C07214=1045.953,107.180,-87.113,170.483,36.346,156.840
C07215=1045.947,106.931,-87.093,170.482,36.345,156.840
C07216=1045.940,106.682,-87.073,170.480,36.343,156.840
C07217=1045.935,106.432,-87.053,170.478,36.342,156.840
C07218=1045.928,106.184,-87.034,170.477,36.340,156.839
C07219=1045.922,105.935,-87.014,170.474,36.338,156.839
C07220=1045.916,105.685,-86.994,170.472,36.337,156.839
C07221=1045.910,105.436,-86.974,170.470,36.335,156.838
C07222=1045.904,105.187,-86.955,170.469,36.334,156.838
C07223=1045.898,104.938,-86.935,170.467,36.332,156.838
C07224=1045.891,104.688,-86.916,170.465,36.331,156.838
C07225=1045.885,104.439,-86.896,170.463,36.330,156.837
C07226=1045.879,104.190,-86.876,170.461,36.328,156.837
C07227=1045.873,103.941,-86.856,170.459,36.327,156.837
C07228=1045.867,103.692,-86.837,170.458,36.325,156.836
C07229=1045.860,103.443,-86.817,170.456,36.323,156.836
C07230=1045.854,103.193,-86.798,170.454,36.322,156.836
C07231=1045.848,102.944,-86.778,170.452,36.320,156.835
C07232=1045.842,102.696,-86.758,170.450,36.318,156.835
C07233=1045.837,102.446,-86.739,170.448,36.317,156.835
C07234=1045.831,102.197,-86.719,170.447,36.316,156.835
C07235=1045.823,101.948,-86.700,170.445,36.314,156.834
C07236=1045.817,101.699,-86.680,170.443,36.313,156.834
C07237=1045.812,101.449,-86.661,170.441,36.311,156.834
C07238=1045.806,101.201,-86.641,170.439,36.310,156.833
C07239=1045.800,100.951,-86.622,170.437,36.308,156.833
C07240=1045.793,100.703,-86.602,170.436,36.307,156.833
C07241=1045.787,100.452,-86.583,170.434,36.305,156.833
C07242=1045.781,100.204,-86.563,170.432,36.303,156.832
C07243=1045.775,99.955,-86.544,170.430,36.302,156.832
C07244=1045.769,99.705,-86.525,170.428,36.300,156.832
C07245=1045.762,99.457,-86.505,170.426,36.299,156.831
C07246=1045.756,99.206,-86.486,170.425,36.298,156.831
C07247=1045.750,98.958,-86.466,170.423,36.296,156.831
C07248=1045.744,98.708,-86.447,170.421,36.295,156.831
C07249=1045.738,98.459,-86.428,170.419,36.293,156.830
C07250=1045.731,98.211,-86.409,170.417,36.292,156.830
C07251=1045.725,97.961,-86.389,170.415,36.290,156.830
C07252=1045.719,97.712,-86.371,170.413,36.289,156.830
C07253=1045.712,97.462,-86.350,170.412,36.287,156.829
C07254=1045.706,97.213,-86.332,170.410,36.286,156.829
C07255=1045.700,96.965,-86.312,170.408,36.284,156.829
C07256=1045.694,96.715,-86.293,170.406,36.283,156.828
C07257=1045.688,96.466,-86.274,170.404,36.282,156.828
C07258=1045.682,96.217,-86.255,170.402,36.280,156.828
C07259=1045.675,95.968,-86.235,170.401,36.278,156.828
C07260=1045.670,95.719,-86.216,170.399,36.277,156.827
C07261=1045.663,95.469,-86.197,170.397,36.275,156.827
C07262=1045.657,95.220,-86.177,170.395,36.274,156.827
C07263=1045.650,94.971,-86.158,170.393,36.273,156.827
C07264=1045.645,94.721,-86.139,170.391,36.271,156.826
C07265=1045.638,94.472,-86.121,170.390,36.270,156.826
C07266=1045.632,94.224,-86.101,170.388,36.268,156.826
C07267=1045.626,93.974,-86.082,170.386,36.266,156.825
C07268=1045.618,93.627,-86.055,170.383,36.265,156.825
C07269=1045.609,93.280,-86.028,170.381,36.262,156.824
C07270=1045.600,92.933,-86.001,170.378,36.260,156.824
C07271=1045.592,92.585,-85.975,170.376,36.258,156.824
C07272=1045.586,92.337,-85.955,170.374,36.256,156.823
C07273=1045.580,92.087,-85.937,170.372,36.255,156.823
C07274=1045.574,91.838,-85.918,170.370,36.254,156.823
C07275=1045.567,91.589,-85.899,170.368,36.252,156.823
C07276=1045.562,91.339,-85.880,170.367,36.251,156.822
C07277=1045.555,91.090,-85.861,170.365,36.249,156.822
C07278=1045.549,90.841,-85.841,170.363,36.248,156.822
C07279=1045.543,90.592,-85.822,170.362,36.246,156.822
C07280=1045.537,90.343,-85.803,170.359,36.245,156.821
C07281=1045.531,90.094,-85.784,170.357,36.243,156.821
C07282=1045.524,89.845,-85.766,170.356,36.242,156.821
C07283=1045.518,89.596,-85.747,170.354,36.240,156.820
C07284=1045.512,89.345,-85.728,170.352,36.239,156.820
C07285=1045.505,89.096,-85.709,170.351,36.238,156.820
C07286=1045.499,88.847,-85.690,170.349,36.236,156.820
C07287=1045.493,88.598,-85.671,170.346,36.234,156.819
C07288=1045.487,88.349,-85.652,170.345,36.233,156.819
C07289=1045.480,88.099,-85.634,170.343,36.232,156.819
C07290=1045.474,87.850,-85.615,170.341,36.231,156.819
C07291=1045.467,87.601,-85.596,170.340,36.229,156.818
C07292=1045.462,87.352,-85.577,170.338,36.228,156.818
C07293=1045.455,87.103,-85.559,170.335,36.226,156.818
C07294=1045.449,86.854,-85.540,170.334,36.224,156.817
C07295=1045.442,86.604,-85.521,170.332,36.223,156.817
C07296=1045.437,86.355,-85.502,170.330,36.222,156.817
C07297=1045.430,86.106,-85.483,170.329,36.221,156.817
C07298=1045.424,85.857,-85.465,170.327,36.219,156.816
C07299=1045.418,85.608,-85.446,170.325,36.217,156.816
C07300=1045.412,85.358,-85.427,170.323,36.216,156.816
C07301=1045.405,85.109,-85.408,170.321,36.214,156.816
C07302=1045.399,84.860,-85.390,170.319,36.213,156.815
C07303=1045.393,84.611,-85.371,170.318,36.212,156.815
C07304=1045.387,84.361,-85.352,170.316,36.211,156.815
C07305=1045.380,84.112,-85.333,170.314,36.209,156.815
C07306=1045.374,83.863,-85.315,170.313,36.207,156.814
C07307=1045.368,83.614,-85.297,170.310,36.206,156.814
C07308=1045.362,83.365,-85.278,170.308,36.204,156.814
C07309=1045.356,83.116,-85.259,170.307,36.203,156.813
C07310=1045.350,82.866,-85.240,170.305,36.202,156.813
C07311=1045.344,82.617,-85.222,170.303,36.200,156.813
C07312=1045.337,82.368,-85.203,170.302,36.199,156.813
C07313=1045.331,82.118,-85.185,170.300,36.197,156.812
C07314=1045.325,81.869,-85.166,170.297,36.195,156.812
C07315=1045.319,81.620,-85.147,170.296,36.194,156.812
C07316=1045.312,81.371,-85.128,170.294,36.193,156.812
C07317=1045.306,81.122,-85.110,170.292,36.192,156.811
C07318=1045.300,80.873,-85.091,170.291,36.190,156.811
C07319=1045.295,80.623,-85.073,170.289,36.188,156.811
C07320=1045.288,80.374,-85.054,170.288,36.187,156.811
C07321=1045.282,80.125,-85.036,170.285,36.185,156.810
C07322=1045.276,79.876,-85.017,170.283,36.184,156.810
C07323=1045.269,79.626,-84.999,170.282,36.183,156.810
C07324=1045.264,79.408,-84.982,170.280,36.181,156.809
C07325=1045.259,79.189,-84.966,170.279,36.180,156.809
C07326=1045.254,78.971,-84.950,170.277,36.178,156.809
C07327=1045.248,78.752,-84.934,170.275,36.177,156.809
C07328=1045.243,78.533,-84.917,170.273,36.176,156.808
C07329=1045.237,78.314,-84.901,170.272,36.175,156.808
C07330=1045.231,78.096,-84.885,170.270,36.173,156.808
C07331=1045.227,77.877,-84.869,170.269,36.172,156.808
C07332=1045.219,77.591,-84.848,170.267,36.171,156.807
C07333=1045.212,77.306,-84.827,170.265,36.169,156.807
C07334=1045.205,77.019,-84.806,170.263,36.168,156.807
C07335=1045.198,76.733,-84.785,170.260,36.166,156.807
C07336=1045.192,76.484,-84.766,170.259,36.164,156.806
C07337=1045.185,76.235,-84.748,170.257,36.163,156.806
C07338=1045.179,75.985,-84.730,170.255,36.161,156.806
C07339=1045.173,75.736,-84.711,170.254,36.160,156.805
C07340=1045.167,75.487,-84.693,170.252,36.159,156.805
C07341=1045.160,75.237,-84.675,170.250,36.158,156.805
C07342=1045.154,74.988,-84.657,170.248,36.156,156.805
C07343=1045.148,74.739,-84.638,170.246,36.154,156.804
C07344=1045.142,74.490,-84.620,170.244,36.153,156.804
C07345=1045.135,74.241,-84.602,170.243,36.152,156.804
C07346=1045.129,73.992,-84.584,170.241,36.151,156.804
C07347=1045.122,73.742,-84.566,170.239,36.149,156.803
C07348=1045.117,73.494,-84.548,170.238,36.147,156.803
C07349=1045.111,73.244,-84.530,170.235,36.146,156.803
C07350=1045.104,72.995,-84.511,170.233,36.145,156.803
C07351=1045.098,72.745,-84.493,170.232,36.143,156.802
C07352=1045.092,72.496,-84.474,170.230,36.142,156.802
C07353=1045.085,72.246,-84.456,170.228,36.140,156.802
C07354=1045.080,71.998,-84.438,170.227,36.139,156.802
C07355=1045.073,71.748,-84.420,170.225,36.137,156.801
C07356=1045.067,71.499,-84.402,170.222,36.136,156.801
C07357=1045.060,71.249,-84.384,170.221,36.135,156.801
C07358=1045.054,71.001,-84.366,170.219,36.134,156.801
C07359=1045.048,70.751,-84.348,170.217,36.132,156.800
C07360=1045.042,70.502,-84.329,170.216,36.130,156.800
C07361=1045.036,70.252,-84.311,170.214,36.129,156.800
C07362=1045.030,70.003,-84.294,170.213,36.128,156.800
C07363=1045.024,69.754,-84.275,170.210,36.126,156.799
C07364=1045.018,69.504,-84.257,170.208,36.125,156.799
C07365=1045.010,69.256,-84.239,170.207,36.123,156.799
C07366=1045.004,69.006,-84.221,170.205,36.122,156.799
C07367=1044.999,68.757,-84.204,170.203,36.121,156.798
C07368=1044.992,68.508,-84.185,170.202,36.119,156.798
C07369=1044.986,68.258,-84.168,170.200,36.118,156.798
C07370=1044.979,68.009,-84.150,170.197,36.116,156.797
C07371=1044.974,67.760,-84.132,170.196,36.115,156.797
C07372=1044.967,67.510,-84.114,170.194,36.114,156.797
C07373=1044.961,67.261,-84.096,170.192,36.112,156.797
C07374=1044.954,67.012,-84.078,170.191,36.111,156.796
C07375=1044.949,66.763,-84.060,170.189,36.109,156.796
C07376=1044.943,66.513,-84.042,170.187,36.108,156.796
C07377=1044.935,66.264,-84.024,170.186,36.107,156.796
C07378=1044.930,66.015,-84.006,170.183,36.106,156.795
C07379=1044.924,65.765,-83.989,170.181,36.104,156.795
C07380=1044.917,65.516,-83.971,170.180,36.102,156.795
C07381=1044.910,65.267,-83.953,170.178,36.101,156.795
C07382=1044.905,65.018,-83.935,170.176,36.100,156.794
C07383=1044.898,64.768,-83.918,170.174,36.099,156.794
C07384=1044.892,64.519,-83.900,170.173,36.097,156.794
C07385=1044.886,64.270,-83.881,170.170,36.095,156.794
C07386=1044.880,64.020,-83.864,170.168,36.094,156.793
C07387=1044.873,63.771,-83.846,170.167,36.093,156.793
C07388=1044.866,63.522,-83.829,170.165,36.092,156.793
C07389=1044.861,63.273,-83.811,170.163,36.090,156.793
C07390=1044.854,63.023,-83.794,170.162,36.089,156.792
C07391=1044.848,62.773,-83.776,170.160,36.088,156.792
C07392=1044.841,62.525,-83.758,170.158,36.087,156.792
C07393=1044.835,62.276,-83.740,170.156,36.085,156.792
C07394=1044.828,62.026,-83.723,170.154,36.084,156.792
C07395=1044.822,61.776,-83.705,170.152,36.083,156.791
C07396=1044.814,61.491,-83.686,170.150,36.081,156.791
C07397=1044.807,61.204,-83.665,170.148,36.080,156.791
C07398=1044.800,60.918,-83.645,170.146,36.078,156.791
C07399=1044.792,60.632,-83.625,170.144,36.076,156.790
C07400=1044.787,60.383,-83.608,170.142,36.075,156.790
C07401=1044.780,60.133,-83.590,170.140,36.074,156.790
C07402=1044.773,59.884,-83.573,170.138,36.073,156.789
C07403=1044.768,59.635,-83.555,170.137,36.071,156.789
C07404=1044.760,59.386,-83.537,170.135,36.070,156.789
C07405=1044.754,59.136,-83.519,170.133,36.069,156.789
C07406=1044.748,58.887,-83.502,170.132,36.067,156.789
C07407=1044.742,58.638,-83.484,170.130,36.066,156.788
C07408=1044.735,58.388,-83.467,170.128,36.065,156.788
C07409=1044.729,58.139,-83.450,170.126,36.063,156.788
C07410=1044.723,57.890,-83.432,170.124,36.062,156.788
C07411=1044.716,57.641,-83.415,170.122,36.060,156.787
C07412=1044.711,57.391,-83.398,170.120,36.059,156.787
C07413=1044.704,57.141,-83.381,170.119,36.058,156.787
C07414=1044.698,56.892,-83.364,170.117,36.057,156.787
C07415=1044.691,56.643,-83.346,170.115,36.055,156.786
C07416=1044.685,56.393,-83.328,170.113,36.054,156.786
C07417=1044.679,56.144,-83.311,170.111,36.053,156.786
C07418=1044.672,55.895,-83.294,170.109,36.052,156.786
C07419=1044.666,55.646,-83.277,170.108,36.050,156.785
C07420=1044.660,55.396,-83.259,170.106,36.048,156.785
C07421=1044.653,55.147,-83.241,170.104,36.047,156.785
C07422=1044.647,54.898,-83.224,170.103,36.046,156.785
C07423=1044.641,54.648,-83.206,170.101,36.045,156.784
C07424=1044.634,54.400,-83.189,170.098,36.043,156.784
C07425=1044.628,54.149,-83.172,170.097,36.042,156.784
C07426=1044.622,53.901,-83.155,170.095,36.041,156.784
C07427=1044.615,53.651,-83.138,170.093,36.039,156.783
C07428=1044.610,53.402,-83.120,170.091,36.038,156.783
C07429=1044.603,53.153,-83.103,170.090,36.037,156.783
C07430=1044.596,52.903,-83.086,170.088,36.035,156.783
C07431=1044.591,52.654,-83.068,170.086,36.034,156.782
C07432=1044.584,52.404,-83.051,170.084,36.032,156.782
C07433=1044.579,52.155,-83.034,170.082,36.031,156.782
C07434=1044.572,51.906,-83.017,170.080,36.030,156.782
C07435=1044.565,51.657,-83.000,170.079,36.029,156.782
C07436=1044.559,51.407,-82.982,170.077,36.027,156.781
C07437=1044.553,51.158,-82.965,170.075,36.026,156.781
C07438=1044.546,50.908,-82.948,170.074,36.024,156.781
C07439=1044.541,50.659,-82.930,170.072,36.023,156.780
C07440=1044.534,50.410,-82.913,170.069,36.022,156.780
C07441=1044.528,50.161,-82.897,170.068,36.020,156.780
C07442=1044.522,49.911,-82.879,170.066,36.019,156.780
C07443=1044.516,49.662,-82.862,170.064,36.018,156.780
C07444=1044.509,49.413,-82.845,170.063,36.016,156.779
C07445=1044.504,49.163,-82.828,170.061,36.015,156.779
C07446=1044.497,48.914,-82.810,170.059,36.013,156.779
C07447=1044.491,48.665,-82.793,170.057,36.012,156.779
C07448=1044.485,48.416,-82.776,170.055,36.011,156.778
C07449=1044.479,48.166,-82.759,170.053,36.009,156.778
C07450=1044.472,47.917,-82.742,170.051,36.008,156.778
C07451=1044.466,47.667,-82.724,170.050,36.007,156.778
C07452=1044.460,47.418,-82.708,170.048,36.006,156.777
C07453=1044.453,47.169,-82.691,170.046,36.004,156.777
C07454=1044.448,46.920,-82.673,170.045,36.002,156.777
C07455=1044.441,46.670,-82.657,170.043,36.001,156.777
C07456=1044.435,46.421,-82.640,170.040,36.000,156.776
C07457=1044.429,46.172,-82.622,170.039,35.999,156.776
C07458=1044.423,45.922,-82.605,170.037,35.997,156.776
C07459=1044.417,45.673,-82.588,170.035,35.996,156.776
C07460=1044.410,45.386,-82.569,170.033,35.994,156.775
C07461=1044.402,45.100,-82.549,170.031,35.993,156.775
C07462=1044.396,44.813,-82.530,170.029,35.991,156.775
C07463=1044.389,44.527,-82.510,170.027,35.990,156.775
C07464=1044.382,44.277,-82.493,170.025,35.988,156.774
C07465=1044.376,44.029,-82.476,170.023,35.986,156.774
C07466=1044.371,43.779,-82.459,170.021,35.985,156.774
C07467=1044.364,43.529,-82.442,170.020,35.984,156.774
C07468=1044.358,43.280,-82.426,170.018,35.983,156.773
C07469=1044.351,43.031,-82.408,170.016,35.981,156.773
C07470=1044.345,42.781,-82.392,170.015,35.980,156.773
C07471=1044.340,42.532,-82.375,170.013,35.979,156.773
C07472=1044.333,42.282,-82.358,170.010,35.977,156.772
C07473=1044.327,42.033,-82.341,170.009,35.976,156.772
C07474=1044.320,41.783,-82.324,170.007,35.975,156.772
C07475=1044.314,41.535,-82.307,170.005,35.974,156.772
C07476=1044.308,41.285,-82.291,170.003,35.972,156.771
C07477=1044.301,41.036,-82.274,170.002,35.971,156.771
C07478=1044.295,40.787,-82.257,170.000,35.970,156.771
C07479=1044.289,40.536,-82.241,169.998,35.968,156.771
C07480=1044.283,40.288,-82.224,169.996,35.967,156.770
C07481=1044.277,40.038,-82.208,169.994,35.965,156.770
C07482=1044.270,39.789,-82.190,169.992,35.964,156.770
C07483=1044.264,39.540,-82.174,169.990,35.963,156.770
C07484=1044.258,39.290,-82.158,169.989,35.961,156.770
C07485=1044.251,39.041,-82.140,169.987,35.960,156.769
C07486=1044.245,38.792,-82.124,169.985,35.959,156.769
C07487=1044.239,38.543,-82.107,169.984,35.958,156.769
C07488=1044.232,38.293,-82.091,169.981,35.956,156.769
C07489=1044.227,38.043,-82.074,169.979,35.955,156.768
C07490=1044.221,37.794,-82.057,169.977,35.954,156.768
C07491=1044.214,37.544,-82.040,169.976,35.952,156.768
C07492=1044.207,37.295,-82.024,169.974,35.951,156.768
C07493=1044.202,37.046,-82.008,169.972,35.950,156.767
C07494=1044.195,36.796,-81.991,169.970,35.949,156.767
C07495=1044.189,36.547,-81.975,169.969,35.947,156.767
C07496=1044.183,36.298,-81.958,169.967,35.946,156.767
C07497=1044.176,36.048,-81.941,169.964,35.945,156.767
C07498=1044.170,35.799,-81.925,169.962,35.943,156.766
C07499=1044.163,35.550,-81.909,169.961,35.942,156.766
C07500=1044.157,35.300,-81.893,169.959,35.942,156.766
C07501=1044.151,35.051,-81.876,169.957,35.940,156.766
C07502=1044.144,34.802,-81.859,169.956,35.939,156.766
C07503=1044.138,34.552,-81.843,169.954,35.938,156.765
C07504=1044.132,34.302,-81.826,169.952,35.936,156.765
C07505=1044.125,34.053,-81.811,169.950,35.935,156.765
C07506=1044.119,33.803,-81.794,169.948,35.934,156.765
C07507=1044.112,33.555,-81.777,169.946,35.933,156.764
C07508=1044.107,33.305,-81.761,169.944,35.931,156.764
C07509=1044.101,33.056,-81.745,169.942,35.930,156.764
C07510=1044.093,32.806,-81.729,169.941,35.929,156.764
C07511=1044.087,32.557,-81.712,169.939,35.927,156.763
C07512=1044.081,32.308,-81.696,169.937,35.926,156.763
C07513=1044.075,32.059,-81.679,169.935,35.925,156.763
C07514=1044.069,31.809,-81.662,169.934,35.924,156.763
C07515=1044.062,31.560,-81.647,169.931,35.922,156.763
C07516=1044.056,31.310,-81.631,169.929,35.921,156.762
C07517=1044.050,31.061,-81.614,169.927,35.920,156.762
C07518=1044.043,30.811,-81.598,169.926,35.918,156.762
C07519=1044.037,30.562,-81.581,169.924,35.917,156.762
C07520=1044.031,30.313,-81.566,169.922,35.916,156.761
C07521=1044.025,30.063,-81.550,169.920,35.914,156.761
C07522=1044.018,29.813,-81.533,169.919,35.914,156.761
C07523=1044.012,29.564,-81.516,169.917,35.913,156.761
C07524=1044.005,29.278,-81.498,169.914,35.911,156.761
C07525=1043.998,28.991,-81.479,169.912,35.909,156.760
C07526=1043.991,28.705,-81.460,169.910,35.908,156.760
C07527=1043.984,28.418,-81.442,169.908,35.907,156.760
C07528=1043.978,28.169,-81.426,169.906,35.905,156.760
C07529=1043.971,27.919,-81.410,169.904,35.904,156.759
C07530=1043.965,27.669,-81.394,169.903,35.903,156.759
C07531=1043.958,27.420,-81.378,169.901,35.902,156.759
C07532=1043.952,27.171,-81.362,169.899,35.900,156.759
C07533=1043.946,26.922,-81.345,169.896,35.899,156.759
C07534=1043.939,26.672,-81.329,169.895,35.898,156.758
C07535=1043.933,26.423,-81.313,169.893,35.896,156.758
C07536=1043.927,26.173,-81.297,169.891,35.896,156.758
C07537=1043.920,25.924,-81.281,169.889,35.894,156.758
C07538=1043.914,25.675,-81.265,169.887,35.893,156.757
C07539=1043.907,25.425,-81.249,169.886,35.892,156.757
C07540=1043.901,25.176,-81.233,169.884,35.891,156.757
C07541=1043.894,24.927,-81.217,169.882,35.889,156.757
C07542=1043.889,24.677,-81.202,169.879,35.888,156.757
C07543=1043.883,24.427,-81.185,169.878,35.887,156.756
C07544=1043.876,24.178,-81.170,169.876,35.886,156.756
C07545=1043.869,23.928,-81.153,169.874,35.885,156.756
C07546=1043.863,23.679,-81.137,169.872,35.883,156.756
C07547=1043.857,23.430,-81.121,169.870,35.882,156.756
C07548=1043.850,23.181,-81.105,169.869,35.881,156.755
C07549=1043.844,22.931,-81.090,169.867,35.880,156.755
C07550=1043.839,22.682,-81.074,169.865,35.879,156.755
C07551=1043.832,22.433,-81.058,169.863,35.878,156.755
C07552=1043.825,22.183,-81.041,169.861,35.876,156.755
C07553=1043.819,21.934,-81.026,169.859,35.875,156.754
C07554=1043.813,21.684,-81.010,169.857,35.874,156.754
C07555=1043.806,21.434,-80.994,169.855,35.872,156.754
C07556=1043.800,21.185,-80.978,169.853,35.871,156.754
C07557=1043.794,20.936,-80.963,169.852,35.870,156.753
C07558=1043.788,20.686,-80.947,169.850,35.869,156.753
C07559=1043.781,20.437,-80.931,169.848,35.868,156.753
C07560=1043.775,20.188,-80.915,169.846,35.867,156.753
C07561=1043.769,19.938,-80.899,169.844,35.865,156.753
C07562=1043.762,19.688,-80.884,169.842,35.864,156.752
C07563=1043.756,19.439,-80.868,169.840,35.863,156.752
C07564=1043.750,19.190,-80.852,169.838,35.861,156.752
C07565=1043.743,18.940,-80.837,169.836,35.861,156.752
C07566=1043.737,18.691,-80.820,169.834,35.859,156.752
C07567=1043.731,18.442,-80.805,169.833,35.858,156.751
C07568=1043.724,18.192,-80.790,169.831,35.857,156.751
C07569=1043.718,17.943,-80.774,169.829,35.856,156.751
C07570=1043.712,17.694,-80.758,169.827,35.855,156.751
C07571=1043.706,17.444,-80.742,169.825,35.854,156.751
C07572=1043.699,17.195,-80.727,169.823,35.852,156.750
C07573=1043.693,16.946,-80.711,169.821,35.851,156.750
C07574=1043.687,16.696,-80.695,169.819,35.850,156.750
C07575=1043.680,16.447,-80.680,169.817,35.849,156.750
C07576=1043.675,16.197,-80.664,169.815,35.848,156.750
C07577=1043.668,15.948,-80.649,169.814,35.847,156.749
C07578=1043.661,15.698,-80.633,169.812,35.845,156.749
C07579=1043.655,15.448,-80.617,169.810,35.844,156.749
C07580=1043.648,15.199,-80.601,169.808,35.843,156.749
C07581=1043.643,14.949,-80.586,169.806,35.842,156.749
C07582=1043.636,14.700,-80.570,169.804,35.841,156.748
C07583=1043.630,14.450,-80.555,169.802,35.839,156.748
C07584=1043.624,14.201,-80.539,169.800,35.838,156.748
C07585=1043.617,13.951,-80.524,169.798,35.837,156.748
C07586=1043.611,13.702,-80.508,169.796,35.836,156.748
C07587=1043.604,13.452,-80.493,169.794,35.835,156.747
C07588=1043.597,13.167,-80.476,169.792,35.834,156.747
C07589=1043.589,12.882,-80.458,169.790,35.832,156.747
C07590=1043.582,12.597,-80.441,169.788,35.831,156.747
C07591=1043.575,12.312,-80.422,169.786,35.830,156.747
C07592=1043.569,12.062,-80.408,169.784,35.829,156.746
C07593=1043.562,11.813,-80.392,169.781,35.828,156.746
C07594=1043.556,11.564,-80.377,169.779,35.827,156.746
C07595=1043.550,11.314,-80.362,169.778,35.826,156.746
C07596=1043.543,11.065,-80.346,169.776,35.824,156.746
C07597=1043.537,10.815,-80.331,169.774,35.823,156.745
C07598=1043.531,10.566,-80.315,169.772,35.822,156.745
C07599=1043.524,10.316,-80.300,169.770,35.821,156.745
C07600=1043.518,10.067,-80.285,169.768,35.820,156.745
C07601=1043.511,9.818,-80.270,169.766,35.819,156.745
C07602=1043.505,9.568,-80.255,169.765,35.818,156.745
C07603=1043.498,9.318,-80.240,169.762,35.817,156.744
C07604=1043.492,9.069,-80.224,169.760,35.816,156.744
C07605=1043.485,8.820,-80.209,169.758,35.815,156.744
C07606=1043.480,8.570,-80.194,169.756,35.813,156.744
C07607=1043.473,8.321,-80.178,169.754,35.813,156.744
C07608=1043.467,8.071,-80.163,169.752,35.811,156.743
C07609=1043.460,7.821,-80.148,169.751,35.810,156.743
C07610=1043.453,7.572,-80.132,169.749,35.809,156.743
C07611=1043.447,7.323,-80.117,169.747,35.808,156.743
C07612=1043.441,7.073,-80.102,169.745,35.807,156.743
C07613=1043.435,6.824,-80.088,169.743,35.806,156.743
C07614=1043.428,6.575,-80.072,169.741,35.805,156.742
C07615=1043.422,6.325,-80.057,169.738,35.803,156.742
C07616=1043.416,6.075,-80.042,169.737,35.803,156.742
C07617=1043.410,5.826,-80.027,169.735,35.801,156.742
C07618=1043.403,5.577,-80.011,169.733,35.800,156.742
C07619=1043.397,5.327,-79.996,169.731,35.799,156.741
C07620=1043.390,5.077,-79.981,169.729,35.798,156.741
C07621=1043.384,4.828,-79.966,169.727,35.797,156.741
C07622=1043.378,4.579,-79.952,169.725,35.796,156.741
C07623=1043.372,4.330,-79.936,169.724,35.795,156.741
C07624=1043.365,4.080,-79.921,169.722,35.794,156.740
C07625=1043.359,3.830,-79.906,169.720,35.792,156.740
C07626=1043.352,3.581,-79.891,169.717,35.792,156.740
C07627=1043.347,3.331,-79.876,169.715,35.790,156.740
C07628=1043.340,3.081,-79.861,169.713,35.789,156.740
C07629=1043.334,2.833,-79.845,169.711,35.788,156.740
C07630=1043.328,2.583,-79.830,169.709,35.787,156.739
C07631=1043.322,2.333,-79.815,169.708,35.786,156.739
C07632=1043.315,2.084,-79.801,169.706,35.785,156.739
C07633=1043.309,1.834,-79.786,169.704,35.784,156.739
C07634=1043.303,1.585,-79.771,169.702,35.783,156.739
C07635=1043.297,1.335,-79.756,169.700,35.781,156.738
C07636=1043.290,1.086,-79.741,169.698,35.781,156.738
C07637=1043.284,0.837,-79.725,169.695,35.779,156.738
C07638=1043.277,0.587,-79.710,169.693,35.778,156.738
C07639=1043.271,0.338,-79.696,169.692,35.777,156.738
C07640=1043.265,0.088,-79.681,169.690,35.776,156.737
C07641=1043.259,-0.161,-79.666,169.688,35.775,156.737
C07642=1043.252,-0.411,-79.651,169.686,35.774,156.737
C07643=1043.246,-0.661,-79.636,169.684,35.773,156.737
C07644=1043.241,-0.910,-79.621,169.682,35.771,156.737
C07645=1043.234,-1.159,-79.606,169.680,35.771,156.737
C07646=1043.228,-1.409,-79.591,169.678,35.769,156.736
C07647=1043.222,-1.659,-79.576,169.677,35.768,156.736
C07648=1043.216,-1.908,-79.562,169.675,35.767,156.736
C07649=1043.209,-2.157,-79.547,169.672,35.766,156.736
C07650=1043.203,-2.407,-79.532,169.670,35.765,156.736
C07651=1043.197,-2.656,-79.517,169.668,35.763,156.735
C07652=1043.190,-2.939,-79.501,169.666,35.762,156.735
C07653=1043.182,-3.223,-79.483,169.664,35.762,156.735
C07654=1043.176,-3.507,-79.466,169.662,35.760,156.735
C07655=1043.169,-3.790,-79.450,169.659,35.759,156.735
C07656=1043.162,-4.040,-79.436,169.657,35.758,156.734
C07657=1043.156,-4.289,-79.421,169.655,35.757,156.734
C07658=1043.150,-4.538,-79.406,169.654,35.756,156.734
C07659=1043.143,-4.788,-79.391,169.652,35.755,156.734
C07660=1043.136,-5.037,-79.377,169.649,35.754,156.734
C07661=1043.130,-5.286,-79.362,169.647,35.753,156.734
C07662=1043.124,-5.536,-79.348,169.645,35.752,156.733
C07663=1043.118,-5.786,-79.333,169.643,35.751,156.733
C07664=1043.111,-6.035,-79.319,169.641,35.750,156.733
C07665=1043.105,-6.284,-79.304,169.639,35.749,156.733
C07666=1043.098,-6.534,-79.289,169.637,35.748,156.733
C07667=1043.092,-6.784,-79.276,169.635,35.747,156.733
C07668=1043.086,-7.033,-79.261,169.633,35.746,156.732
C07669=1043.080,-7.283,-79.246,169.631,35.745,156.732
C07670=1043.073,-7.532,-79.231,169.629,35.744,156.732
C07671=1043.066,-7.782,-79.217,169.627,35.743,156.732
C07672=1043.061,-8.031,-79.203,169.625,35.742,156.732
C07673=1043.054,-8.281,-79.188,169.623,35.741,156.732
C07674=1043.047,-8.530,-79.174,169.620,35.740,156.731
C07675=1043.042,-8.780,-79.160,169.619,35.739,156.731
C07676=1043.035,-9.029,-79.145,169.617,35.738,156.731
C07677=1043.028,-9.279,-79.130,169.615,35.737,156.731
C07678=1043.022,-9.528,-79.116,169.613,35.736,156.731
C07679=1043.016,-9.778,-79.102,169.611,35.735,156.731
C07680=1043.010,-10.028,-79.087,169.609,35.734,156.730
C07681=1043.003,-10.276,-79.073,169.607,35.733,156.730
C07682=1042.997,-10.527,-79.058,169.605,35.732,156.730
C07683=1042.991,-10.776,-79.044,169.603,35.731,156.730
C07684=1042.984,-11.025,-79.029,169.601,35.730,156.730
C07685=1042.978,-11.275,-79.015,169.599,35.729,156.730
C07686=1042.972,-11.524,-79.001,169.597,35.728,156.729
C07687=1042.965,-11.774,-78.986,169.594,35.727,156.729
C07688=1042.959,-12.024,-78.972,169.592,35.726,156.729
C07689=1042.953,-12.273,-78.958,169.590,35.725,156.729
C07690=1042.947,-12.523,-78.944,169.588,35.724,156.729
C07691=1042.941,-12.772,-78.929,169.586,35.723,156.729
C07692=1042.934,-13.021,-78.914,169.584,35.722,156.728
C07693=1042.928,-13.271,-78.901,169.582,35.721,156.728
C07694=1042.922,-13.520,-78.886,169.580,35.720,156.728
C07695=1042.916,-13.771,-78.872,169.578,35.719,156.728
C07696=1042.909,-14.019,-78.858,169.576,35.718,156.728
C07697=1042.903,-14.269,-78.843,169.574,35.717,156.728
C07698=1042.897,-14.518,-78.829,169.573,35.716,156.728
C07699=1042.890,-14.768,-78.815,169.571,35.715,156.727
C07700=1042.885,-15.017,-78.801,169.568,35.714,156.727
C07701=1042.878,-15.267,-78.786,169.566,35.713,156.727
C07702=1042.872,-15.517,-78.772,169.564,35.713,156.727
C07703=1042.865,-15.766,-78.758,169.562,35.711,156.727
C07704=1042.859,-16.016,-78.744,169.560,35.711,156.727
C07705=1042.853,-16.264,-78.730,169.558,35.710,156.727
C07706=1042.846,-16.515,-78.716,169.556,35.709,156.726
C07707=1042.840,-16.765,-78.702,169.554,35.708,156.726
C07708=1042.834,-17.014,-78.688,169.552,35.707,156.726
C07709=1042.827,-17.264,-78.674,169.550,35.706,156.726
C07710=1042.820,-17.512,-78.660,169.548,35.705,156.726
C07711=1042.814,-17.763,-78.646,169.546,35.704,156.726
C07712=1042.808,-18.012,-78.633,169.544,35.703,156.725
C07713=1042.802,-18.262,-78.618,169.542,35.702,156.725
C07714=1042.796,-18.511,-78.604,169.540,35.702,156.725
C07715=1042.789,-18.760,-78.589,169.537,35.700,156.725
C07716=1042.782,-19.043,-78.574,169.534,35.700,156.725
C07717=1042.775,-19.324,-78.558,169.532,35.698,156.725
C07718=1042.768,-19.606,-78.542,169.530,35.698,156.725
C07719=1042.761,-19.888,-78.527,169.527,35.696,156.724
C07720=1042.754,-20.137,-78.513,169.525,35.696,156.724
C07721=1042.748,-20.386,-78.499,169.523,35.694,156.724
C07722=1042.742,-20.636,-78.485,169.521,35.694,156.724
C07723=1042.735,-20.885,-78.471,169.519,35.693,156.724
C07724=1042.729,-21.135,-78.457,169.517,35.692,156.724
C07725=1042.723,-21.385,-78.444,169.515,35.691,156.724
C07726=1042.717,-21.635,-78.430,169.513,35.690,156.723
C07727=1042.710,-21.884,-78.416,169.511,35.689,156.723
C07728=1042.703,-22.133,-78.402,169.509,35.688,156.723
C07729=1042.698,-22.383,-78.388,169.507,35.688,156.723
C07730=1042.691,-22.633,-78.374,169.504,35.686,156.723
C07731=1042.684,-22.882,-78.360,169.502,35.686,156.723
C07732=1042.678,-23.132,-78.346,169.500,35.685,156.723
C07733=1042.672,-23.381,-78.333,169.498,35.684,156.722
C07734=1042.667,-23.631,-78.319,169.496,35.683,156.722
C07735=1042.660,-23.880,-78.305,169.494,35.682,156.722
C07736=1042.653,-24.129,-78.291,169.492,35.681,156.722
C07737=1042.647,-24.380,-78.277,169.490,35.680,156.722
C07738=1042.641,-24.629,-78.264,169.488,35.680,156.722
C07739=1042.635,-24.878,-78.251,169.486,35.679,156.722
C07740=1042.628,-25.128,-78.236,169.484,35.678,156.721
C07741=1042.622,-25.377,-78.222,169.482,35.677,156.721
C07742=1042.615,-25.627,-78.209,169.480,35.676,156.721
C07743=1042.610,-25.877,-78.195,169.478,35.675,156.721
C07744=1042.604,-26.126,-78.182,169.476,35.674,156.721
C07745=1042.598,-26.376,-78.167,169.474,35.674,156.721
C07746=1042.591,-26.625,-78.154,169.471,35.672,156.721
C07747=1042.585,-26.874,-78.140,169.469,35.672,156.720
C07748=1042.578,-27.124,-78.127,169.467,35.671,156.720
C07749=1042.573,-27.374,-78.113,169.464,35.670,156.720
C07750=1042.566,-27.624,-78.099,169.462,35.669,156.720
C07751=1042.560,-27.873,-78.086,169.460,35.668,156.720
C07752=1042.553,-28.122,-78.073,169.458,35.668,156.720
C07753=1042.547,-28.372,-78.059,169.456,35.667,156.720
C07754=1042.540,-28.621,-78.046,169.454,35.666,156.720
C07755=1042.534,-28.871,-78.032,169.452,35.666,156.720
C07756=1042.527,-29.121,-78.019,169.450,35.664,156.719
C07757=1042.522,-29.370,-78.005,169.448,35.664,156.719
C07758=1042.515,-29.620,-77.991,169.446,35.663,156.719
C07759=1042.509,-29.869,-77.978,169.444,35.662,156.719
C07760=1042.503,-30.119,-77.965,169.442,35.661,156.719
C07761=1042.496,-30.369,-77.951,169.440,35.661,156.719
C07762=1042.490,-30.618,-77.938,169.437,35.659,156.719
C07763=1042.483,-30.867,-77.925,169.435,35.659,156.718
C07764=1042.477,-31.117,-77.911,169.432,35.658,156.718
C07765=1042.470,-31.366,-77.898,169.430,35.657,156.718
C07766=1042.464,-31.616,-77.885,169.428,35.657,156.718
C07767=1042.458,-31.867,-77.871,169.426,35.656,156.718
C07768=1042.452,-32.116,-77.858,169.424,35.655,156.718
C07769=1042.446,-32.365,-77.844,169.422,35.654,156.718
C07770=1042.439,-32.615,-77.831,169.420,35.653,156.718
C07771=1042.433,-32.864,-77.817,169.418,35.653,156.718
C07772=1042.427,-33.114,-77.804,169.416,35.652,156.717
C07773=1042.420,-33.363,-77.791,169.413,35.651,156.717
C07774=1042.414,-33.613,-77.777,169.411,35.651,156.717
C07775=1042.408,-33.863,-77.765,169.409,35.650,156.717
C07776=1042.402,-34.112,-77.751,169.407,35.649,156.717
C07777=1042.395,-34.361,-77.738,169.405,35.648,156.717
C07778=1042.389,-34.611,-77.724,169.403,35.647,156.717
C07779=1042.382,-34.860,-77.711,169.401,35.647,156.717
C07780=1042.376,-35.142,-77.696,169.398,35.646,156.716
C07781=1042.369,-35.422,-77.681,169.396,35.644,156.716
C07782=1042.362,-35.704,-77.666,169.394,35.644,156.716
C07783=1042.354,-35.985,-77.651,169.390,35.643,156.716
C07784=1042.348,-36.234,-77.638,169.388,35.642,156.716
C07785=1042.342,-36.484,-77.625,169.386,35.642,156.716
C07786=1042.336,-36.733,-77.612,169.384,35.641,156.716
C07787=1042.330,-36.982,-77.599,169.382,35.640,156.716
C07788=1042.323,-37.232,-77.585,169.380,35.639,156.715
C07789=1042.317,-37.482,-77.573,169.378,35.638,156.715
C07790=1042.311,-37.732,-77.559,169.376,35.638,156.715
C07791=1042.305,-37.981,-77.546,169.373,35.637,156.715
C07792=1042.299,-38.231,-77.534,169.371,35.636,156.715
C07793=1042.292,-38.481,-77.520,169.369,35.636,156.715
C07794=1042.286,-38.730,-77.507,169.367,35.635,156.715
C07795=1042.280,-38.980,-77.494,169.365,35.634,156.715
C07796=1042.274,-39.229,-77.481,169.363,35.634,156.715
C07797=1042.267,-39.478,-77.468,169.361,35.633,156.715
C07798=1042.261,-39.729,-77.455,169.358,35.632,156.714
C07799=1042.255,-39.978,-77.441,169.356,35.631,156.714
C07800=1042.248,-40.227,-77.429,169.354,35.631,156.714
C07801=1042.242,-40.477,-77.416,169.352,35.630,156.714
C07802=1042.236,-40.726,-77.403,169.350,35.629,156.714
C07803=1042.229,-40.977,-77.390,169.348,35.629,156.714
C07804=1042.223,-41.226,-77.377,169.345,35.628,156.714
C07805=1042.216,-41.476,-77.365,169.342,35.627,156.714
C07806=1042.210,-41.725,-77.352,169.340,35.627,156.714
C07807=1042.204,-41.974,-77.338,169.338,35.626,156.714
C07808=1042.198,-42.224,-77.326,169.336,35.625,156.713
C07809=1042.192,-42.473,-77.312,169.334,35.625,156.713
C07810=1042.184,-42.724,-77.300,169.332,35.624,156.713
C07811=1042.178,-42.973,-77.287,169.329,35.623,156.713
C07812=1042.172,-43.223,-77.274,169.327,35.622,156.713
C07813=1042.166,-43.472,-77.261,169.325,35.622,156.713
C07814=1042.160,-43.722,-77.248,169.323,35.621,156.713
C07815=1042.153,-43.971,-77.236,169.321,35.621,156.713
C07816=1042.147,-44.221,-77.223,169.319,35.620,156.713
C07817=1042.141,-44.470,-77.210,169.316,35.620,156.713
C07818=1042.135,-44.720,-77.197,169.314,35.619,156.713
C07819=1042.128,-44.970,-77.184,169.312,35.618,156.712
C07820=1042.122,-45.219,-77.172,169.310,35.618,156.712
C07821=1042.116,-45.469,-77.159,169.308,35.617,156.712
C07822=1042.110,-45.719,-77.146,169.306,35.616,156.712
C07823=1042.104,-45.969,-77.133,169.303,35.615,156.712
C07824=1042.097,-46.217,-77.121,169.301,35.615,156.712
C07825=1042.091,-46.467,-77.108,169.299,35.614,156.712
C07826=1042.085,-46.717,-77.096,169.297,35.613,156.712
C07827=1042.079,-46.967,-77.082,169.295,35.613,156.712
C07828=1042.072,-47.216,-77.070,169.291,35.612,156.711
C07829=1042.066,-47.465,-77.057,169.290,35.612,156.712
C07830=1042.060,-47.715,-77.045,169.287,35.611,156.711
C07831=1042.054,-47.965,-77.032,169.285,35.611,156.711
C07832=1042.047,-48.214,-77.019,169.283,35.610,156.711
C07833=1042.041,-48.464,-77.007,169.281,35.609,156.711
C07834=1042.035,-48.714,-76.994,169.278,35.609,156.711
C07835=1042.029,-48.963,-76.981,169.276,35.608,156.711
C07836=1042.022,-49.213,-76.969,169.274,35.607,156.711
C07837=1042.016,-49.463,-76.956,169.272,35.606,156.711
C07838=1042.010,-49.712,-76.943,169.270,35.606,156.711
C07839=1042.004,-49.961,-76.931,169.267,35.605,156.710
C07840=1041.998,-50.211,-76.919,169.265,35.605,156.711
C07841=1041.992,-50.461,-76.906,169.263,35.604,156.710
C07842=1041.985,-50.710,-76.893,169.261,35.604,156.710
C07843=1041.979,-50.960,-76.881,169.259,35.603,156.710
C07844=1041.972,-51.242,-76.867,169.256,35.603,156.710
C07845=1041.964,-51.523,-76.853,169.254,35.602,156.710
C07846=1041.957,-51.805,-76.840,169.251,35.601,156.710
C07847=1041.950,-52.086,-76.826,169.248,35.601,156.710
C07848=1041.943,-52.335,-76.814,169.246,35.601,156.710
C07849=1041.937,-52.585,-76.801,169.244,35.600,156.710
C07850=1041.931,-52.835,-76.789,169.242,35.599,156.710
C07851=1041.925,-53.084,-76.776,169.239,35.599,156.710
C07852=1041.918,-53.334,-76.764,169.237,35.599,156.710
C07853=1041.911,-53.583,-76.752,169.235,35.598,156.710
C07854=1041.905,-53.833,-76.739,169.233,35.598,156.710
C07855=1041.899,-54.083,-76.727,169.230,35.597,156.709
C07856=1041.892,-54.332,-76.715,169.228,35.596,156.709
C07857=1041.886,-54.582,-76.703,169.226,35.596,156.709
C07858=1041.880,-54.832,-76.691,169.224,35.596,156.709
C07859=1041.874,-55.082,-76.678,169.221,35.596,156.709
C07860=1041.867,-55.331,-76.666,169.219,35.595,156.709
C07861=1041.860,-55.581,-76.654,169.216,35.594,156.709
C07862=1041.854,-55.831,-76.642,169.214,35.594,156.709
C07863=1041.848,-56.080,-76.630,169.211,35.593,156.709
C07864=1041.841,-56.330,-76.618,169.209,35.593,156.709
C07865=1041.835,-56.580,-76.605,169.207,35.593,156.709
C07866=1041.829,-56.829,-76.593,169.205,35.592,156.709
C07867=1041.823,-57.078,-76.582,169.202,35.592,156.709
C07868=1041.817,-57.328,-76.569,169.200,35.591,156.709
C07869=1041.810,-57.578,-76.557,169.198,35.591,156.709
C07870=1041.804,-57.828,-76.545,169.196,35.591,156.709
C07871=1041.797,-58.077,-76.533,169.193,35.590,156.709
C07872=1041.791,-58.327,-76.521,169.191,35.589,156.708
C07873=1041.785,-58.577,-76.508,169.189,35.589,156.708
C07874=1041.778,-58.826,-76.496,169.187,35.588,156.708
C07875=1041.772,-59.075,-76.485,169.184,35.588,156.708
C07876=1041.766,-59.325,-76.472,169.182,35.588,156.708
C07877=1041.760,-59.574,-76.460,169.180,35.587,156.708
C07878=1041.753,-59.824,-76.448,169.177,35.587,156.708
C07879=1041.747,-60.074,-76.436,169.175,35.586,156.708
C07880=1041.740,-60.323,-76.424,169.173,35.586,156.708
C07881=1041.734,-60.574,-76.413,169.171,35.585,156.708
C07882=1041.729,-60.823,-76.400,169.168,35.585,156.708
C07883=1041.722,-61.072,-76.388,169.166,35.585,156.708
C07884=1041.715,-61.322,-76.376,169.164,35.584,156.708
C07885=1041.710,-61.572,-76.364,169.161,35.584,156.708
C07886=1041.703,-61.821,-76.352,169.159,35.583,156.708
C07887=1041.697,-62.070,-76.340,169.157,35.583,156.708
C07888=1041.691,-62.321,-76.329,169.155,35.582,156.708
C07889=1041.685,-62.570,-76.317,169.152,35.582,156.708
C07890=1041.678,-62.820,-76.305,169.150,35.582,156.708
C07891=1041.671,-63.070,-76.293,169.148,35.581,156.707
C07892=1041.666,-63.319,-76.280,169.146,35.581,156.707
C07893=1041.660,-63.569,-76.269,169.143,35.580,156.707
C07894=1041.653,-63.818,-76.257,169.141,35.580,156.707
C07895=1041.647,-64.068,-76.245,169.139,35.579,156.707
C07896=1041.641,-64.317,-76.233,169.136,35.579,156.707
C07897=1041.635,-64.567,-76.222,169.134,35.579,156.707
C07898=1041.628,-64.817,-76.210,169.132,35.578,156.707
C07899=1041.622,-65.067,-76.197,169.129,35.578,156.707
C07900=1041.616,-65.316,-76.186,169.127,35.577,156.707
C07901=1041.610,-65.566,-76.174,169.125,35.577,156.707
C07902=1041.604,-65.816,-76.162,169.123,35.577,156.707
C07903=1041.598,-66.065,-76.150,169.120,35.576,156.707
C07904=1041.592,-66.315,-76.139,169.118,35.576,156.707
C07905=1041.585,-66.564,-76.127,169.116,35.576,156.707
C07906=1041.580,-66.814,-76.115,169.113,35.575,156.707
C07907=1041.573,-67.064,-76.104,169.111,35.575,156.707
C07908=1041.566,-67.346,-76.090,169.108,35.574,156.707
C07909=1041.559,-67.629,-76.077,169.105,35.574,156.707
C07910=1041.552,-67.912,-76.064,169.103,35.573,156.707
C07911=1041.545,-68.195,-76.051,169.100,35.573,156.706
C07912=1041.539,-68.444,-76.039,169.097,35.573,156.707
C07913=1041.533,-68.693,-76.026,169.095,35.572,156.706
C07914=1041.527,-68.944,-76.015,169.093,35.572,156.706
C07915=1041.520,-69.193,-76.003,169.090,35.571,156.706
C07916=1041.515,-69.443,-75.992,169.088,35.571,156.706
C07917=1041.509,-69.693,-75.980,169.086,35.570,156.706
C07918=1041.502,-69.942,-75.968,169.084,35.570,156.706
C07919=1041.496,-70.192,-75.957,169.081,35.570,156.706
C07920=1041.490,-70.441,-75.945,169.079,35.570,156.706
C07921=1041.485,-70.691,-75.934,169.077,35.569,156.706
C07922=1041.478,-70.941,-75.922,169.074,35.569,156.706
C07923=1041.472,-71.191,-75.910,169.072,35.568,156.706
C07924=1041.466,-71.440,-75.899,169.070,35.568,156.706
C07925=1041.460,-71.690,-75.887,169.067,35.567,156.706
C07926=1041.454,-71.939,-75.875,169.065,35.567,156.706
C07927=1041.448,-72.189,-75.864,169.063,35.567,156.706
C07928=1041.441,-72.439,-75.852,169.060,35.567,156.706
C07929=1041.435,-72.688,-75.841,169.058,35.566,156.706
C07930=1041.429,-72.938,-75.829,169.056,35.566,156.706
C07931=1041.424,-73.188,-75.818,169.053,35.565,156.706
C07932=1041.417,-73.437,-75.806,169.051,35.565,156.706
C07933=1041.411,-73.687,-75.795,169.049,35.564,156.706
C07934=1041.406,-73.937,-75.783,169.046,35.564,156.706
C07935=1041.400,-74.186,-75.772,169.044,35.564,156.706
C07936=1041.393,-74.436,-75.760,169.042,35.564,156.705
C07937=1041.386,-74.685,-75.749,169.039,35.563,156.705
C07938=1041.380,-74.935,-75.738,169.037,35.563,156.706
C07939=1041.374,-75.185,-75.727,169.035,35.563,156.705
C07940=1041.368,-75.434,-75.715,169.032,35.563,156.705
C07941=1041.361,-75.684,-75.704,169.030,35.563,156.705
C07942=1041.356,-75.934,-75.693,169.028,35.563,156.705
C07943=1041.349,-76.183,-75.681,169.025,35.562,156.705
C07944=1041.343,-76.433,-75.670,169.023,35.562,156.705
C07945=1041.337,-76.683,-75.659,169.020,35.562,156.705
C07946=1041.331,-76.933,-75.648,169.018,35.562,156.705
C07947=1041.325,-77.182,-75.636,169.016,35.561,156.705
C07948=1041.318,-77.432,-75.625,169.013,35.561,156.705
C07949=1041.313,-77.682,-75.614,169.011,35.561,156.705
C07950=1041.306,-77.931,-75.602,169.009,35.561,156.705
C07951=1041.300,-78.181,-75.591,169.006,35.560,156.705
C07952=1041.294,-78.431,-75.580,169.004,35.560,156.705
C07953=1041.288,-78.680,-75.569,169.002,35.560,156.705
C07954=1041.282,-78.931,-75.558,168.999,35.560,156.705
C07955=1041.276,-79.180,-75.546,168.997,35.559,156.705
C07956=1041.269,-79.430,-75.535,168.994,35.559,156.705
C07957=1041.263,-79.679,-75.525,168.992,35.559,156.705
C07958=1041.256,-79.929,-75.514,168.990,35.559,156.705
C07959=1041.251,-80.179,-75.503,168.987,35.559,156.705
C07960=1041.244,-80.429,-75.491,168.985,35.559,156.705
C07961=1041.238,-80.677,-75.480,168.982,35.559,156.705
C07962=1041.231,-80.928,-75.469,168.980,35.558,156.705
C07963=1041.226,-81.177,-75.458,168.978,35.558,156.705
C07964=1041.219,-81.427,-75.447,168.975,35.558,156.705
C07965=1041.213,-81.676,-75.437,168.973,35.558,156.705
C07966=1041.206,-81.927,-75.426,168.970,35.558,156.705
C07967=1041.201,-82.176,-75.415,168.968,35.558,156.705
C07968=1041.194,-82.425,-75.404,168.966,35.558,156.705
C07969=1041.188,-82.675,-75.393,168.963,35.558,156.705
C07970=1041.182,-82.925,-75.382,168.961,35.558,156.705
C07971=1041.175,-83.175,-75.372,168.958,35.558,156.705
C07972=1041.168,-83.459,-75.359,168.956,35.558,156.705
C07973=1041.161,-83.744,-75.346,168.953,35.557,156.705
C07974=1041.154,-84.030,-75.334,168.950,35.557,156.705
C07975=1041.147,-84.314,-75.322,168.947,35.557,156.705
C07976=1041.140,-84.564,-75.311,168.945,35.557,156.705
C07977=1041.135,-84.814,-75.300,168.942,35.557,156.705
C07978=1041.129,-85.063,-75.289,168.940,35.557,156.705
C07979=1041.122,-85.313,-75.279,168.938,35.557,156.705
C07980=1041.116,-85.563,-75.268,168.935,35.557,156.705
C07981=1041.110,-85.813,-75.257,168.933,35.557,156.705
C07982=1041.103,-86.062,-75.246,168.930,35.557,156.705
C07983=1041.097,-86.312,-75.235,168.928,35.557,156.705
C07984=1041.091,-86.562,-75.224,168.925,35.557,156.706
C07985=1041.085,-86.811,-75.214,168.923,35.557,156.706
C07986=1041.079,-87.060,-75.203,168.921,35.557,156.706
C07987=1041.073,-87.311,-75.192,168.918,35.557,156.706
C07988=1041.066,-87.560,-75.182,168.916,35.557,156.706
C07989=1041.060,-87.810,-75.170,168.913,35.556,156.706
C07990=1041.053,-88.059,-75.160,168.911,35.556,156.706
C07991=1041.048,-88.309,-75.150,168.908,35.556,156.706
C07992=1041.042,-88.559,-75.139,168.906,35.556,156.706
C07993=1041.035,-88.809,-75.128,168.904,35.556,156.706
C07994=1041.029,-89.058,-75.117,168.901,35.556,156.706
C07995=1041.023,-89.308,-75.107,168.899,35.556,156.706
C07996=1041.016,-89.557,-75.096,168.896,35.556,156.706
C07997=1041.011,-89.808,-75.086,168.894,35.556,156.706
C07998=1041.005,-90.057,-75.075,168.891,35.556,156.706
C07999=1040.998,-90.307,-75.064,168.889,35.556,156.706
C08000=1040.992,-90.556,-75.053,168.886,35.556,156.706
C08001=1040.986,-90.806,-75.043,168.884,35.556,156.706
C08002=1040.981,-91.056,-75.033,168.882,35.556,156.706
C08003=1040.974,-91.306,-75.022,168.879,35.556,156.706
C08004=1040.968,-91.555,-75.011,168.877,35.556,156.706
C08005=1040.962,-91.805,-75.001,168.874,35.556,156.706
C08006=1040.956,-92.054,-74.991,168.872,35.556,156.706
C08007=1040.949,-92.305,-74.980,168.869,35.556,156.706
C08008=1040.944,-92.554,-74.969,168.868,35.556,156.706
C08009=1040.937,-92.803,-74.959,168.865,35.556,156.706
C08010=1040.932,-93.053,-74.948,168.863,35.556,156.706
C08011=1040.925,-93.303,-74.938,168.861,35.556,156.706
C08012=1040.919,-93.553,-74.927,168.858,35.556,156.706
C08013=1040.914,-93.803,-74.917,168.856,35.556,156.706
C08014=1040.907,-94.052,-74.906,168.853,35.556,156.706
C08015=1040.901,-94.302,-74.896,168.851,35.556,156.706
C08016=1040.895,-94.552,-74.886,168.848,35.556,156.706
C08017=1040.889,-94.802,-74.875,168.846,35.556,156.706
C08018=1040.882,-95.051,-74.864,168.843,35.556,156.706
C08019=1040.877,-95.301,-74.854,168.841,35.556,156.706
C08020=1040.871,-95.550,-74.843,168.839,35.556,156.706
C08021=1040.865,-95.799,-74.833,168.836,35.556,156.706
C08022=1040.859,-96.050,-74.823,168.834,35.556,156.706
C08023=1040.852,-96.299,-74.812,168.831,35.556,156.706
C08024=1040.847,-96.550,-74.802,168.829,35.556,156.706
C08025=1040.840,-96.799,-74.792,168.826,35.556,156.706
C08026=1040.835,-97.048,-74.781,168.824,35.556,156.706
C08027=1040.829,-97.298,-74.771,168.821,35.556,156.706
C08028=1040.823,-97.548,-74.761,168.819,35.557,156.707
C08029=1040.816,-97.798,-74.751,168.816,35.557,156.707
C08030=1040.810,-98.048,-74.740,168.814,35.557,156.707
C08031=1040.804,-98.297,-74.730,168.811,35.556,156.707
C08032=1040.797,-98.546,-74.720,168.809,35.557,156.707
C08033=1040.792,-98.797,-74.710,168.806,35.557,156.707
C08034=1040.786,-99.046,-74.699,168.804,35.557,156.707
C08035=1040.779,-99.296,-74.690,168.801,35.558,156.707
C08036=1040.773,-99.583,-74.678,168.799,35.557,156.707
C08037=1040.765,-99.870,-74.666,168.796,35.558,156.707
C08038=1040.758,-100.157,-74.655,168.793,35.558,156.707
C08039=1040.751,-100.445,-74.643,168.790,35.558,156.707
C08040=1040.745,-100.694,-74.633,168.787,35.558,156.707
C08041=1040.739,-100.944,-74.623,168.785,35.558,156.707
C08042=1040.733,-101.194,-74.613,168.782,35.558,156.707
C08043=1040.727,-101.443,-74.603,168.780,35.559,156.707
C08044=1040.720,-101.694,-74.593,168.777,35.559,156.707
C08045=1040.714,-101.943,-74.582,168.775,35.559,156.708
C08046=1040.708,-102.193,-74.572,168.772,35.559,156.708
C08047=1040.702,-102.443,-74.563,168.770,35.559,156.708
C08048=1040.696,-102.692,-74.552,168.767,35.560,156.708
C08049=1040.690,-102.942,-74.542,168.765,35.560,156.708
C08050=1040.684,-103.192,-74.533,168.762,35.560,156.708
C08051=1040.677,-103.441,-74.523,168.760,35.560,156.708
C08052=1040.672,-103.691,-74.512,168.757,35.560,156.708
C08053=1040.666,-103.941,-74.503,168.756,35.561,156.708
C08054=1040.660,-104.191,-74.493,168.753,35.561,156.708
C08055=1040.653,-104.440,-74.483,168.751,35.561,156.708
C08056=1040.648,-104.690,-74.473,168.748,35.561,156.708
C08057=1040.641,-104.940,-74.463,168.746,35.561,156.708
C08058=1040.635,-105.189,-74.453,168.743,35.562,156.708
C08059=1040.629,-105.439,-74.443,168.741,35.562,156.708
C08060=1040.623,-105.689,-74.433,168.738,35.562,156.708
C08061=1040.617,-105.939,-74.424,168.736,35.562,156.708
C08062=1040.611,-106.188,-74.413,168.733,35.563,156.709
C08063=1040.605,-106.438,-74.404,168.731,35.563,156.709
C08064=1040.599,-106.688,-74.394,168.728,35.563,156.709
C08065=1040.593,-106.938,-74.384,168.726,35.563,156.709
C08066=1040.587,-107.187,-74.374,168.723,35.564,156.709
C08067=1040.581,-107.437,-74.365,168.721,35.564,156.709
C08068=1040.574,-107.686,-74.355,168.718,35.565,156.709
C08069=1040.568,-107.936,-74.345,168.716,35.564,156.709
C08070=1040.562,-108.186,-74.335,168.713,35.565,156.709
C08071=1040.556,-108.436,-74.325,168.711,35.565,156.709
C08072=1040.550,-108.686,-74.316,168.708,35.566,156.709
C08073=1040.544,-108.936,-74.306,168.706,35.566,156.709
C08074=1040.538,-109.185,-74.297,168.703,35.566,156.709
C08075=1040.532,-109.435,-74.287,168.701,35.567,156.710
C08076=1040.525,-109.684,-74.277,168.698,35.567,156.710
C08077=1040.519,-109.934,-74.267,168.695,35.567,156.710
C08078=1040.513,-110.184,-74.258,168.693,35.567,156.710
C08079=1040.507,-110.434,-74.248,168.690,35.568,156.710
C08080=1040.501,-110.684,-74.239,168.688,35.568,156.710
C08081=1040.495,-110.933,-74.229,168.685,35.568,156.710
C08082=1040.489,-111.182,-74.220,168.684,35.569,156.710
C08083=1040.483,-111.432,-74.210,168.681,35.569,156.710
C08084=1040.476,-111.682,-74.201,168.679,35.569,156.710
C08085=1040.471,-111.932,-74.190,168.676,35.570,156.710
C08086=1040.465,-112.182,-74.181,168.674,35.570,156.710
C08087=1040.459,-112.432,-74.171,168.671,35.570,156.711
C08088=1040.452,-112.682,-74.162,168.668,35.571,156.711
C08089=1040.446,-112.931,-74.152,168.666,35.571,156.711
C08090=1040.441,-113.180,-74.143,168.663,35.572,156.711
C08091=1040.435,-113.430,-74.133,168.661,35.572,156.711
C08092=1040.428,-113.680,-74.124,168.658,35.572,156.711
C08093=1040.422,-113.930,-74.114,168.656,35.573,156.711
C08094=1040.416,-114.180,-74.105,168.653,35.573,156.711
C08095=1040.410,-114.430,-74.096,168.651,35.573,156.711
C08096=1040.404,-114.680,-74.086,168.648,35.574,156.711
C08097=1040.398,-114.929,-74.077,168.646,35.574,156.711
C08098=1040.392,-115.179,-74.068,168.643,35.575,156.712
C08099=1040.386,-115.429,-74.058,168.640,35.575,156.712
C08100=1040.379,-115.715,-74.048,168.637,35.576,156.712
C08101=1040.372,-116.001,-74.037,168.635,35.576,156.712
C08102=1040.365,-116.287,-74.025,168.632,35.577,156.712
C08103=1040.357,-116.574,-74.015,168.629,35.577,156.712
C08104=1040.352,-116.823,-74.006,168.627,35.578,156.712
C08105=1040.346,-117.073,-73.997,168.625,35.578,156.712
C08106=1040.340,-117.323,-73.987,168.622,35.578,156.712
C08107=1040.334,-117.573,-73.978,168.619,35.579,156.712
C08108=1040.328,-117.823,-73.968,168.617,35.580,156.713
C08109=1040.322,-118.072,-73.959,168.614,35.580,156.713
C08110=1040.315,-118.322,-73.951,168.612,35.580,156.713
///RCONF 1,0,0,0,1,0,0,0,0,0,0,0,0,0,0,0,0,0,0,0,0,0,0,0
C08111=1040.309,-118.572,-73.941,168.609,35.581,156.713
C08112=1040.303,-118.821,-73.932,168.607,35.581,156.713
C08113=1040.297,-119.071,-73.922,168.604,35.582,156.713
C08114=1040.292,-119.321,-73.914,168.601,35.582,156.713
C08115=1040.285,-119.571,-73.904,168.599,35.583,156.713
C08116=1040.279,-119.821,-73.894,168.596,35.583,156.713
C08117=1040.273,-120.070,-73.887,168.594,35.584,156.714
C08118=1040.267,-120.320,-73.877,168.591,35.584,156.714
C08119=1040.261,-120.570,-73.867,168.589,35.585,156.714
C08120=1040.255,-120.819,-73.858,168.586,35.585,156.714
C08121=1040.249,-121.069,-73.849,168.583,35.586,156.714
C08122=1040.243,-121.319,-73.840,168.581,35.587,156.714
C08123=1040.236,-121.568,-73.831,168.579,35.587,156.714
C08124=1040.230,-121.819,-73.822,168.577,35.587,156.714
C08125=1040.225,-122.068,-73.813,168.574,35.588,156.714
C08126=1040.219,-122.318,-73.804,168.571,35.588,156.715
C08127=1040.213,-122.568,-73.794,168.569,35.589,156.715
C08128=1040.207,-122.817,-73.785,168.566,35.589,156.715
C08129=1040.201,-123.067,-73.777,168.564,35.590,156.715
C08130=1040.195,-123.317,-73.767,168.561,35.591,156.715
C08131=1040.189,-123.567,-73.759,168.559,35.591,156.715
C08132=1040.183,-123.817,-73.749,168.556,35.592,156.715
C08133=1040.176,-124.066,-73.740,168.553,35.592,156.715
C08134=1040.170,-124.316,-73.731,168.551,35.593,156.716
C08135=1040.165,-124.566,-73.722,168.548,35.594,156.716
C08136=1040.159,-124.816,-73.713,168.546,35.594,156.716
C08137=1040.152,-125.065,-73.704,168.543,35.595,156.716
C08138=1040.147,-125.315,-73.696,168.540,35.595,156.716
C08139=1040.141,-125.565,-73.686,168.538,35.596,156.716
C08140=1040.134,-125.815,-73.678,168.535,35.597,156.716
C08141=1040.128,-126.064,-73.669,168.534,35.597,156.716
C08142=1040.123,-126.315,-73.660,168.531,35.598,156.717
C08143=1040.116,-126.563,-73.651,168.528,35.598,156.717
C08144=1040.110,-126.814,-73.643,168.526,35.599,156.717
C08145=1040.104,-127.064,-73.633,168.523,35.599,156.717
C08146=1040.098,-127.313,-73.625,168.521,35.600,156.717
C08147=1040.092,-127.563,-73.616,168.518,35.601,156.717
C08148=1040.087,-127.813,-73.607,168.515,35.601,156.717
C08149=1040.081,-128.062,-73.598,168.513,35.602,156.717
C08150=1040.076,-128.312,-73.588,168.511,35.602,156.717
C08151=1040.073,-128.562,-73.577,168.508,35.601,156.717
C08152=1040.070,-128.812,-73.567,168.506,35.600,156.717
C08153=1040.067,-129.061,-73.555,168.504,35.598,156.717
C08154=1040.066,-129.312,-73.542,168.503,35.596,156.717
C08155=1040.066,-129.561,-73.529,168.500,35.594,156.716
C08156=1040.066,-129.812,-73.516,168.498,35.591,156.716
C08157=1040.067,-130.061,-73.502,168.497,35.587,156.715
C08158=1040.068,-130.312,-73.487,168.496,35.584,156.715
C08159=1040.072,-130.562,-73.472,168.494,35.579,156.714
C08160=1040.076,-130.812,-73.456,168.493,35.575,156.713
C08161=1040.080,-131.063,-73.439,168.492,35.569,156.712
C08162=1040.085,-131.313,-73.423,168.491,35.563,156.711
C08163=1040.090,-131.562,-73.405,168.490,35.558,156.710
C08164=1039.746,-131.587,-73.665,168.442,35.755,156.744
C08165=1039.739,-131.337,-73.683,168.444,35.761,156.745
C08166=1039.734,-131.087,-73.700,168.444,35.766,156.746
C08167=1039.730,-130.837,-73.716,168.446,35.772,156.747
C08168=1039.726,-130.586,-73.732,168.447,35.777,156.748
C08169=1039.724,-130.336,-73.748,168.448,35.781,156.748
C08170=1039.722,-130.087,-73.763,168.450,35.785,156.749
C08171=1039.720,-129.835,-73.777,168.452,35.788,156.749
C08172=1039.721,-129.585,-73.790,168.453,35.791,156.750
C08173=1039.721,-129.336,-73.804,168.455,35.793,156.750
C08174=1039.722,-129.086,-73.816,168.456,35.795,156.751
C08175=1039.724,-128.836,-73.827,168.459,35.797,156.751
C08176=1039.727,-128.586,-73.838,168.461,35.798,156.751
C08177=1039.731,-128.336,-73.849,168.464,35.799,156.751
C08178=1039.735,-128.086,-73.859,168.466,35.799,156.751
C08179=1039.740,-127.837,-73.869,168.468,35.799,156.751
C08180=1039.746,-127.588,-73.877,168.471,35.798,156.751
C08181=1039.752,-127.338,-73.886,168.473,35.798,156.751
C08182=1039.758,-127.087,-73.895,168.475,35.797,156.751
C08183=1039.765,-126.839,-73.904,168.478,35.796,156.751
C08184=1039.771,-126.588,-73.913,168.480,35.795,156.750
C08185=1039.776,-126.338,-73.921,168.483,35.795,156.750
C08186=1039.783,-126.089,-73.930,168.486,35.794,156.750
C08187=1039.789,-125.839,-73.939,168.488,35.793,156.750
C08188=1039.794,-125.589,-73.948,168.491,35.793,156.750
C08189=1039.801,-125.339,-73.956,168.494,35.792,156.750
C08190=1039.807,-125.090,-73.966,168.496,35.792,156.750
C08191=1039.812,-124.840,-73.974,168.499,35.791,156.750
C08192=1039.819,-124.590,-73.983,168.501,35.790,156.749
C08193=1039.825,-124.340,-73.992,168.504,35.790,156.749
C08194=1039.831,-124.091,-74.001,168.507,35.789,156.749
C08195=1039.837,-123.841,-74.011,168.509,35.789,156.749
C08196=1039.843,-123.591,-74.019,168.512,35.788,156.749
C08197=1039.849,-123.342,-74.028,168.513,35.787,156.749
C08198=1039.855,-123.091,-74.037,168.516,35.787,156.749
C08199=1039.861,-122.842,-74.047,168.519,35.786,156.749
C08200=1039.866,-122.592,-74.055,168.521,35.785,156.748
C08201=1039.873,-122.342,-74.064,168.524,35.785,156.748
C08202=1039.879,-122.093,-74.074,168.526,35.784,156.748
C08203=1039.885,-121.842,-74.083,168.529,35.784,156.748
C08204=1039.891,-121.593,-74.092,168.532,35.783,156.748
C08205=1039.897,-121.343,-74.101,168.534,35.782,156.748
C08206=1039.903,-121.093,-74.110,168.537,35.782,156.748
C08207=1039.909,-120.844,-74.119,168.539,35.781,156.748
C08208=1039.915,-120.594,-74.129,168.542,35.781,156.748
C08209=1039.921,-120.344,-74.137,168.545,35.781,156.747
C08210=1039.927,-120.094,-74.147,168.547,35.780,156.747
C08211=1039.933,-119.845,-74.156,168.550,35.780,156.747
C08212=1039.939,-119.595,-74.164,168.552,35.779,156.747
C08213=1039.946,-119.345,-74.174,168.555,35.778,156.747
C08214=1039.952,-119.095,-74.184,168.558,35.778,156.747
C08215=1039.957,-118.846,-74.193,168.559,35.777,156.747
C08216=1039.963,-118.596,-74.202,168.562,35.776,156.747
C08217=1039.969,-118.346,-74.211,168.564,35.777,156.747
C08218=1039.976,-118.096,-74.221,168.567,35.776,156.746
C08219=1039.982,-117.847,-74.230,168.570,35.775,156.746
C08220=1039.988,-117.597,-74.238,168.572,35.775,156.746
C08221=1039.994,-117.347,-74.248,168.575,35.774,156.746
C08222=1040.000,-117.097,-74.257,168.577,35.774,156.746
C08223=1040.006,-116.848,-74.267,168.580,35.774,156.746
C08224=1040.012,-116.598,-74.276,168.582,35.773,156.746
///RCONF 1,0,0,0,0,0,0,0,0,0,0,0,0,0,0,0,0,0,0,0,0,0,0,0
C08225=1040.019,-116.312,-74.287,168.585,35.772,156.746
C08226=1040.026,-116.026,-74.297,168.588,35.772,156.746
C08227=1040.033,-115.739,-74.308,168.591,35.771,156.745
C08228=1040.039,-115.452,-74.319,168.594,35.771,156.745
C08229=1040.046,-115.203,-74.328,168.597,35.770,156.745
C08230=1040.052,-114.953,-74.337,168.599,35.770,156.745
C08231=1040.058,-114.704,-74.347,168.602,35.769,156.745
C08232=1040.064,-114.454,-74.356,168.605,35.769,156.745
C08233=1040.070,-114.204,-74.366,168.607,35.768,156.745
C08234=1040.077,-113.955,-74.375,168.609,35.768,156.745
C08235=1040.082,-113.704,-74.384,168.611,35.768,156.745
C08236=1040.089,-113.454,-74.394,168.614,35.767,156.745
C08237=1040.095,-113.205,-74.403,168.616,35.766,156.744
C08238=1040.100,-112.956,-74.413,168.619,35.767,156.744
C08239=1040.107,-112.706,-74.422,168.621,35.766,156.744
C08240=1040.112,-112.456,-74.432,168.624,35.765,156.744
C08241=1040.118,-112.206,-74.442,168.627,35.765,156.744
C08242=1040.124,-111.956,-74.451,168.629,35.765,156.744
C08243=1040.130,-111.706,-74.461,168.632,35.764,156.744
C08244=1040.137,-111.456,-74.471,168.634,35.764,156.744
C08245=1040.143,-111.207,-74.480,168.637,35.764,156.744
C08246=1040.149,-110.957,-74.490,168.639,35.763,156.744
C08247=1040.155,-110.708,-74.499,168.642,35.763,156.744
C08248=1040.161,-110.458,-74.508,168.645,35.762,156.744
C08249=1040.167,-110.208,-74.518,168.647,35.762,156.743
C08250=1040.173,-109.958,-74.528,168.650,35.762,156.743
C08251=1040.179,-109.709,-74.537,168.652,35.761,156.743
C08252=1040.186,-109.459,-74.547,168.655,35.761,156.743
C08253=1040.192,-109.210,-74.557,168.657,35.761,156.743
C08254=1040.198,-108.960,-74.567,168.660,35.760,156.743
C08255=1040.203,-108.710,-74.577,168.662,35.760,156.743
C08256=1040.210,-108.460,-74.586,168.665,35.760,156.743
C08257=1040.216,-108.210,-74.596,168.666,35.759,156.743
C08258=1040.222,-107.960,-74.605,168.669,35.759,156.743
C08259=1040.228,-107.710,-74.615,168.672,35.758,156.743
C08260=1040.234,-107.461,-74.625,168.674,35.758,156.742
C08261=1040.241,-107.212,-74.635,168.677,35.758,156.742
C08262=1040.247,-106.962,-74.644,168.679,35.757,156.742
C08263=1040.252,-106.712,-74.655,168.682,35.757,156.742
C08264=1040.259,-106.462,-74.664,168.684,35.757,156.742
C08265=1040.265,-106.212,-74.674,168.687,35.757,156.742
C08266=1040.271,-105.963,-74.684,168.689,35.756,156.742
C08267=1040.277,-105.713,-74.694,168.692,35.756,156.742
C08268=1040.283,-105.463,-74.704,168.694,35.756,156.742
C08269=1040.289,-105.213,-74.713,168.697,35.756,156.742
C08270=1040.296,-104.964,-74.724,168.699,35.755,156.742
C08271=1040.302,-104.714,-74.733,168.702,35.755,156.742
C08272=1040.307,-104.464,-74.743,168.704,35.755,156.742
C08273=1040.313,-104.214,-74.753,168.707,35.755,156.742
C08274=1040.320,-103.965,-74.763,168.710,35.755,156.742
C08275=1040.326,-103.715,-74.773,168.712,35.754,156.742
C08276=1040.331,-103.465,-74.783,168.715,35.754,156.742
C08277=1040.338,-103.216,-74.793,168.717,35.753,156.741
C08278=1040.344,-102.966,-74.803,168.720,35.754,156.741
C08279=1040.349,-102.716,-74.813,168.722,35.753,156.741
C08280=1040.356,-102.467,-74.823,168.725,35.753,156.741
C08281=1040.362,-102.217,-74.833,168.727,35.752,156.741
C08282=1040.368,-101.967,-74.842,168.730,35.752,156.741
C08283=1040.374,-101.718,-74.853,168.732,35.752,156.741
C08284=1040.380,-101.468,-74.863,168.735,35.752,156.741
C08285=1040.386,-101.218,-74.872,168.737,35.752,156.741
C08286=1040.393,-100.968,-74.884,168.740,35.751,156.741
C08287=1040.399,-100.718,-74.893,168.742,35.751,156.741
C08288=1040.405,-100.469,-74.903,168.745,35.751,156.741
C08289=1040.412,-100.181,-74.915,168.747,35.751,156.741
C08290=1040.419,-99.894,-74.926,168.750,35.751,156.741
C08291=1040.426,-99.607,-74.937,168.752,35.750,156.741
C08292=1040.433,-99.320,-74.950,168.755,35.750,156.741
C08293=1040.439,-99.071,-74.959,168.758,35.750,156.740
C08294=1040.446,-98.821,-74.970,168.760,35.750,156.740
C08295=1040.451,-98.571,-74.980,168.763,35.750,156.740
C08296=1040.458,-98.321,-74.991,168.765,35.749,156.740
C08297=1040.464,-98.072,-75.000,168.768,35.749,156.740
C08298=1040.470,-97.822,-75.011,168.770,35.749,156.740
C08299=1040.476,-97.572,-75.021,168.773,35.749,156.740
C08300=1040.482,-97.322,-75.032,168.775,35.749,156.740
C08301=1040.489,-97.072,-75.041,168.778,35.749,156.740
C08302=1040.494,-96.823,-75.052,168.780,35.749,156.740
C08303=1040.500,-96.573,-75.062,168.783,35.748,156.740
C08304=1040.506,-96.324,-75.073,168.785,35.748,156.740
C08305=1040.512,-96.074,-75.082,168.788,35.748,156.740
C08306=1040.518,-95.824,-75.093,168.790,35.748,156.740
C08307=1040.525,-95.575,-75.103,168.793,35.748,156.740
C08308=1040.531,-95.324,-75.114,168.795,35.749,156.740
C08309=1040.536,-95.075,-75.125,168.798,35.748,156.740
C08310=1040.543,-94.826,-75.135,168.800,35.748,156.740
C08311=1040.548,-94.576,-75.145,168.802,35.748,156.740
C08312=1040.555,-94.326,-75.156,168.805,35.748,156.740
C08313=1040.561,-94.076,-75.167,168.807,35.748,156.740
C08314=1040.567,-93.826,-75.176,168.810,35.748,156.740
C08315=1040.573,-93.577,-75.187,168.812,35.748,156.740
C08316=1040.579,-93.327,-75.198,168.815,35.748,156.740
C08317=1040.585,-93.078,-75.208,168.817,35.748,156.740
C08318=1040.591,-92.827,-75.219,168.820,35.748,156.740
C08319=1040.598,-92.578,-75.229,168.822,35.748,156.740
C08320=1040.603,-92.328,-75.239,168.825,35.748,156.740
C08321=1040.609,-92.079,-75.250,168.827,35.748,156.740
C08322=1040.615,-91.829,-75.261,168.830,35.747,156.739
C08323=1040.622,-91.579,-75.272,168.832,35.747,156.739
C08324=1040.628,-91.330,-75.281,168.834,35.747,156.739
C08325=1040.634,-91.080,-75.292,168.837,35.747,156.739
C08326=1040.640,-90.830,-75.303,168.839,35.747,156.739
C08327=1040.646,-90.581,-75.314,168.842,35.748,156.739
C08328=1040.652,-90.331,-75.324,168.844,35.748,156.739
C08329=1040.658,-90.081,-75.335,168.847,35.748,156.739
C08330=1040.665,-89.831,-75.345,168.849,35.748,156.739
C08331=1040.670,-89.582,-75.356,168.852,35.748,156.739
C08332=1040.677,-89.333,-75.367,168.854,35.747,156.739
C08333=1040.683,-89.082,-75.378,168.857,35.747,156.739
C08334=1040.689,-88.832,-75.388,168.859,35.747,156.739
C08335=1040.695,-88.583,-75.398,168.861,35.747,156.739
C08336=1040.701,-88.334,-75.409,168.864,35.747,156.739
C08337=1040.707,-88.083,-75.420,168.866,35.747,156.739
C08338=1040.714,-87.834,-75.431,168.869,35.747,156.739
C08339=1040.719,-87.585,-75.442,168.871,35.747,156.739
C08340=1040.727,-87.335,-75.452,168.874,35.748,156.739
C08341=1040.732,-87.085,-75.462,168.876,35.748,156.739
C08342=1040.738,-86.835,-75.473,168.879,35.748,156.739
C08343=1040.745,-86.585,-75.484,168.881,35.748,156.739
C08344=1040.751,-86.336,-75.495,168.883,35.748,156.739
C08345=1040.757,-86.086,-75.506,168.886,35.747,156.739
C08346=1040.763,-85.836,-75.516,168.887,35.747,156.739
C08347=1040.769,-85.587,-75.527,168.890,35.747,156.739
C08348=1040.775,-85.337,-75.538,168.892,35.747,156.739
C08349=1040.782,-85.088,-75.549,168.895,35.747,156.739
C08350=1040.788,-84.837,-75.560,168.897,35.747,156.739
C08351=1040.794,-84.588,-75.571,168.900,35.747,156.739
C08352=1040.800,-84.339,-75.581,168.902,35.747,156.739
C08353=1040.808,-84.053,-75.593,168.905,35.748,156.739
C08354=1040.815,-83.768,-75.606,168.907,35.748,156.739
C08355=1040.821,-83.484,-75.619,168.910,35.748,156.739
C08356=1040.829,-83.198,-75.631,168.913,35.748,156.739
C08357=1040.835,-82.949,-75.642,168.915,35.748,156.739
C08358=1040.842,-82.699,-75.653,168.918,35.748,156.739
C08359=1040.847,-82.449,-75.664,168.920,35.748,156.739
C08360=1040.854,-82.200,-75.674,168.923,35.748,156.739
C08361=1040.860,-81.950,-75.685,168.925,35.748,156.739
C08362=1040.866,-81.700,-75.696,168.928,35.748,156.739
C08363=1040.873,-81.451,-75.707,168.930,35.748,156.739
C08364=1040.879,-81.201,-75.718,168.932,35.748,156.739
C08365=1040.885,-80.951,-75.729,168.935,35.748,156.739
C08366=1040.891,-80.702,-75.740,168.937,35.748,156.739
C08367=1040.898,-80.452,-75.751,168.940,35.748,156.739
C08368=1040.904,-80.203,-75.762,168.942,35.748,156.739
C08369=1040.910,-79.953,-75.773,168.945,35.748,156.739
C08370=1040.917,-79.703,-75.784,168.947,35.748,156.739
C08371=1040.923,-79.453,-75.795,168.949,35.748,156.739
C08372=1040.929,-79.204,-75.806,168.952,35.749,156.739
C08373=1040.935,-78.954,-75.818,168.954,35.749,156.739
C08374=1040.941,-78.705,-75.828,168.957,35.749,156.739
C08375=1040.948,-78.455,-75.840,168.959,35.749,156.739
C08376=1040.953,-78.205,-75.851,168.961,35.749,156.739
C08377=1040.960,-77.955,-75.863,168.964,35.750,156.739
C08378=1040.966,-77.706,-75.873,168.966,35.750,156.739
C08379=1040.972,-77.456,-75.885,168.968,35.750,156.739
C08380=1040.978,-77.206,-75.896,168.971,35.750,156.739
C08381=1040.984,-76.957,-75.907,168.973,35.750,156.739
C08382=1040.990,-76.707,-75.918,168.976,35.751,156.739
C08383=1040.996,-76.457,-75.930,168.978,35.751,156.739
C08384=1041.003,-76.207,-75.942,168.980,35.751,156.739
C08385=1041.009,-75.958,-75.952,168.983,35.751,156.739
C08386=1041.015,-75.708,-75.964,168.985,35.751,156.739
C08387=1041.021,-75.458,-75.975,168.988,35.752,156.739
C08388=1041.028,-75.209,-75.986,168.990,35.752,156.739
C08389=1041.034,-74.960,-75.997,168.992,35.752,156.739
C08390=1041.041,-74.710,-76.009,168.995,35.752,156.739
C08391=1041.046,-74.460,-76.020,168.997,35.753,156.739
C08392=1041.053,-74.210,-76.031,168.999,35.753,156.739
C08393=1041.059,-73.961,-76.043,169.002,35.753,156.739
C08394=1041.064,-73.711,-76.054,169.004,35.753,156.739
C08395=1041.071,-73.461,-76.066,169.006,35.753,156.739
C08396=1041.077,-73.212,-76.077,169.009,35.753,156.739
C08397=1041.083,-72.962,-76.088,169.011,35.754,156.739
C08398=1041.089,-72.713,-76.100,169.013,35.754,156.739
C08399=1041.095,-72.462,-76.112,169.017,35.755,156.739
C08400=1041.101,-72.213,-76.123,169.019,35.755,156.739
C08401=1041.107,-71.963,-76.135,169.021,35.755,156.739
C08402=1041.114,-71.714,-76.147,169.024,35.756,156.739
C08403=1041.119,-71.464,-76.158,169.026,35.756,156.739
C08404=1041.125,-71.214,-76.170,169.028,35.756,156.739
C08405=1041.131,-70.965,-76.181,169.031,35.756,156.739
C08406=1041.138,-70.715,-76.193,169.033,35.757,156.739
C08407=1041.143,-70.465,-76.205,169.035,35.757,156.739
C08408=1041.149,-70.216,-76.216,169.038,35.758,156.740
C08409=1041.156,-69.966,-76.228,169.040,35.758,156.740
C08410=1041.162,-69.717,-76.239,169.042,35.758,156.739
C08411=1041.169,-69.467,-76.251,169.045,35.759,156.740
C08412=1041.174,-69.217,-76.263,169.047,35.759,156.740
C08413=1041.180,-68.968,-76.275,169.049,35.759,156.740
C08414=1041.187,-68.718,-76.286,169.052,35.759,156.740
C08415=1041.193,-68.468,-76.298,169.054,35.760,156.740
C08416=1041.198,-68.219,-76.310,169.056,35.760,156.740
C08417=1041.206,-67.936,-76.323,169.059,35.761,156.740
C08418=1041.213,-67.653,-76.336,169.062,35.761,156.740
C08419=1041.219,-67.370,-76.349,169.064,35.762,156.740
C08420=1041.226,-67.088,-76.363,169.067,35.762,156.740
C08421=1041.233,-66.838,-76.374,169.069,35.762,156.740
C08422=1041.239,-66.588,-76.386,169.071,35.762,156.740
C08423=1041.245,-66.339,-76.398,169.074,35.763,156.740
C08424=1041.251,-66.089,-76.410,169.076,35.763,156.740
C08425=1041.258,-65.839,-76.422,169.078,35.764,156.740
C08426=1041.263,-65.590,-76.434,169.081,35.764,156.740
C08427=1041.269,-65.340,-76.445,169.083,35.765,156.740
C08428=1041.276,-65.090,-76.457,169.085,35.765,156.740
C08429=1041.283,-64.841,-76.469,169.088,35.765,156.740
C08430=1041.288,-64.592,-76.481,169.090,35.765,156.740
C08431=1041.294,-64.342,-76.492,169.092,35.766,156.741
C08432=1041.301,-64.092,-76.504,169.094,35.766,156.740
C08433=1041.307,-63.842,-76.517,169.097,35.767,156.741
C08434=1041.313,-63.593,-76.529,169.099,35.767,156.741
C08435=1041.319,-63.343,-76.540,169.101,35.768,156.741
C08436=1041.326,-63.093,-76.552,169.104,35.768,156.741
C08437=1041.332,-62.844,-76.564,169.106,35.768,156.741
C08438=1041.338,-62.595,-76.576,169.108,35.768,156.741
C08439=1041.344,-62.345,-76.588,169.111,35.769,156.741
C08440=1041.350,-62.095,-76.600,169.113,35.769,156.741
C08441=1041.357,-61.845,-76.612,169.115,35.770,156.741
C08442=1041.363,-61.595,-76.624,169.117,35.770,156.741
C08443=1041.369,-61.346,-76.636,169.120,35.770,156.741
C08444=1041.375,-61.097,-76.648,169.122,35.770,156.741
C08445=1041.382,-60.847,-76.660,169.124,35.771,156.741
C08446=1041.388,-60.597,-76.672,169.127,35.772,156.741
C08447=1041.394,-60.347,-76.683,169.129,35.772,156.741
C08448=1041.401,-60.097,-76.695,169.131,35.773,156.741
C08449=1041.406,-59.848,-76.708,169.133,35.773,156.741
C08450=1041.413,-59.599,-76.720,169.137,35.773,156.741
C08451=1041.419,-59.349,-76.732,169.139,35.773,156.741
C08452=1041.425,-59.099,-76.744,169.141,35.774,156.742
C08453=1041.432,-58.850,-76.756,169.144,35.774,156.742
C08454=1041.439,-58.600,-76.768,169.146,35.775,156.742
C08455=1041.445,-58.350,-76.781,169.148,35.775,156.742
C08456=1041.451,-58.101,-76.792,169.150,35.776,156.742
C08457=1041.457,-57.851,-76.803,169.153,35.776,156.742
C08458=1041.463,-57.601,-76.816,169.155,35.776,156.742
C08459=1041.469,-57.352,-76.828,169.157,35.777,156.742
C08460=1041.476,-57.102,-76.840,169.160,35.777,156.742
C08461=1041.482,-56.852,-76.852,169.162,35.778,156.742
C08462=1041.489,-56.603,-76.864,169.164,35.778,156.742
C08463=1041.495,-56.353,-76.876,169.166,35.778,156.742
C08464=1041.501,-56.103,-76.889,169.169,35.779,156.742
C08465=1041.508,-55.854,-76.901,169.171,35.779,156.742
C08466=1041.514,-55.605,-76.912,169.173,35.780,156.742
C08467=1041.520,-55.355,-76.925,169.176,35.780,156.742
C08468=1041.527,-55.106,-76.938,169.178,35.781,156.742
C08469=1041.533,-54.856,-76.950,169.180,35.781,156.742
C08470=1041.539,-54.607,-76.962,169.182,35.781,156.742
C08471=1041.546,-54.357,-76.974,169.185,35.782,156.743
C08472=1041.552,-54.107,-76.987,169.187,35.782,156.743
C08473=1041.559,-53.857,-76.999,169.189,35.783,156.743
C08474=1041.565,-53.608,-77.011,169.191,35.783,156.743
C08475=1041.571,-53.358,-77.023,169.194,35.783,156.743
C08476=1041.578,-53.108,-77.035,169.196,35.784,156.743
C08477=1041.584,-52.859,-77.048,169.198,35.784,156.743
C08478=1041.590,-52.609,-77.060,169.200,35.785,156.743
C08479=1041.597,-52.360,-77.072,169.203,35.785,156.743
C08480=1041.603,-52.110,-77.085,169.205,35.786,156.743
C08481=1041.610,-51.828,-77.099,169.207,35.786,156.743
C08482=1041.618,-51.547,-77.112,169.210,35.786,156.743
C08483=1041.625,-51.266,-77.126,169.213,35.787,156.743
C08484=1041.632,-50.984,-77.140,169.215,35.788,156.743
C08485=1041.639,-50.735,-77.152,169.217,35.788,156.743
C08486=1041.645,-50.485,-77.165,169.220,35.788,156.743
C08487=1041.651,-50.236,-77.178,169.222,35.789,156.744
C08488=1041.657,-49.986,-77.190,169.225,35.790,156.744
C08489=1041.663,-49.736,-77.202,169.227,35.790,156.744
C08490=1041.669,-49.486,-77.215,169.229,35.791,156.744
C08491=1041.676,-49.237,-77.228,169.232,35.791,156.744
C08492=1041.682,-48.987,-77.240,169.234,35.792,156.744
C08493=1041.688,-48.737,-77.253,169.236,35.793,156.744
C08494=1041.694,-48.488,-77.266,169.238,35.793,156.744
C08495=1041.701,-48.239,-77.278,169.240,35.794,156.744
C08496=1041.707,-47.989,-77.291,169.243,35.794,156.744
C08497=1041.713,-47.739,-77.304,169.245,35.795,156.744
C08498=1041.719,-47.490,-77.316,169.247,35.795,156.744
C08499=1041.726,-47.240,-77.328,169.249,35.796,156.745
C08500=1041.732,-46.991,-77.342,169.251,35.797,156.745
C08501=1041.738,-46.741,-77.354,169.254,35.797,156.745
C08502=1041.744,-46.492,-77.367,169.256,35.798,156.745
C08503=1041.751,-46.242,-77.379,169.258,35.799,156.745
C08504=1041.757,-45.991,-77.392,169.260,35.799,156.745
C08505=1041.763,-45.742,-77.406,169.262,35.799,156.745
C08506=1041.769,-45.492,-77.418,169.265,35.800,156.745
C08507=1041.776,-45.243,-77.431,169.267,35.801,156.745
C08508=1041.782,-44.993,-77.443,169.269,35.802,156.745
C08509=1041.788,-44.744,-77.457,169.271,35.802,156.745
C08510=1041.794,-44.494,-77.469,169.273,35.803,156.746
C08511=1041.800,-44.245,-77.483,169.275,35.804,156.746
C08512=1041.807,-43.996,-77.494,169.278,35.804,156.746
C08513=1041.813,-43.746,-77.507,169.281,35.804,156.746
C08514=1041.819,-43.496,-77.520,169.283,35.805,156.746
C08515=1041.826,-43.246,-77.533,169.285,35.806,156.746
C08516=1041.833,-42.997,-77.546,169.287,35.806,156.746
C08517=1041.839,-42.747,-77.558,169.290,35.807,156.746
C08518=1041.845,-42.498,-77.572,169.292,35.808,156.746
C08519=1041.851,-42.248,-77.585,169.294,35.808,156.746
C08520=1041.857,-41.999,-77.598,169.296,35.809,156.747
C08521=1041.864,-41.750,-77.610,169.298,35.809,156.746
C08522=1041.870,-41.499,-77.623,169.300,35.810,156.747
C08523=1041.877,-41.250,-77.636,169.303,35.810,156.747
C08524=1041.882,-41.000,-77.649,169.305,35.811,156.747
C08525=1041.889,-40.751,-77.662,169.307,35.812,156.747
C08526=1041.895,-40.501,-77.674,169.309,35.813,156.747
C08527=1041.902,-40.252,-77.687,169.311,35.813,156.747
C08528=1041.908,-40.002,-77.701,169.313,35.814,156.747
C08529=1041.914,-39.752,-77.714,169.316,35.815,156.747
C08530=1041.921,-39.503,-77.727,169.318,35.815,156.747
C08531=1041.927,-39.253,-77.740,169.320,35.815,156.747
C08532=1041.933,-39.004,-77.752,169.322,35.816,156.748
C08533=1041.940,-38.754,-77.766,169.324,35.817,156.748
C08534=1041.946,-38.504,-77.778,169.326,35.817,156.748
C08535=1041.952,-38.255,-77.792,169.328,35.818,156.748
C08536=1041.959,-38.005,-77.805,169.332,35.819,156.748
C08537=1041.965,-37.756,-77.818,169.334,35.819,156.748
C08538=1041.971,-37.506,-77.831,169.336,35.821,156.748
C08539=1041.977,-37.256,-77.844,169.338,35.821,156.748
C08540=1041.984,-37.007,-77.858,169.340,35.822,156.748
C08541=1041.989,-36.757,-77.871,169.342,35.823,156.749
C08542=1041.995,-36.508,-77.884,169.344,35.823,156.749
C08543=1042.002,-36.258,-77.898,169.346,35.824,156.749
C08544=1042.008,-36.008,-77.911,169.349,35.825,156.749
C08545=1042.015,-35.728,-77.925,169.351,35.825,156.749
C08546=1042.023,-35.447,-77.940,169.353,35.826,156.749
C08547=1042.029,-35.165,-77.955,169.356,35.827,156.749
C08548=1042.036,-34.885,-77.970,169.358,35.828,156.749
C08549=1042.043,-34.635,-77.984,169.360,35.829,156.750
C08550=1042.049,-34.386,-77.997,169.362,35.829,156.750
C08551=1042.055,-34.136,-78.009,169.364,35.830,156.750
C08552=1042.062,-33.886,-78.023,169.367,35.831,156.750
C08553=1042.067,-33.636,-78.037,169.369,35.832,156.750
C08554=1042.074,-33.387,-78.050,169.372,35.832,156.750
C08555=1042.080,-33.138,-78.063,169.374,35.833,156.750
C08556=1042.087,-32.888,-78.077,169.376,35.834,156.750
C08557=1042.093,-32.639,-78.090,169.378,35.835,156.750
C08558=1042.099,-32.389,-78.103,169.380,35.836,156.751
C08559=1042.105,-32.139,-78.116,169.382,35.836,156.751
C08560=1042.112,-31.889,-78.130,169.384,35.837,156.751
C08561=1042.118,-31.640,-78.143,169.387,35.838,156.751
C08562=1042.124,-31.391,-78.156,169.389,35.838,156.751
C08563=1042.131,-31.141,-78.170,169.391,35.839,156.751
C08564=1042.137,-30.892,-78.183,169.393,35.840,156.751
C08565=1042.143,-30.642,-78.197,169.395,35.840,156.751
C08566=1042.150,-30.392,-78.211,169.397,35.841,156.751
C08567=1042.156,-30.143,-78.224,169.399,35.842,156.752
C08568=1042.162,-29.894,-78.237,169.401,35.843,156.752
C08569=1042.169,-29.644,-78.251,169.403,35.844,156.752
C08570=1042.175,-29.394,-78.264,169.405,35.844,156.752
C08571=1042.182,-29.144,-78.278,169.408,35.845,156.752
C08572=1042.188,-28.895,-78.291,169.411,35.846,156.752
C08573=1042.194,-28.646,-78.304,169.413,35.846,156.752
C08574=1042.200,-28.396,-78.319,169.415,35.847,156.752
C08575=1042.207,-28.146,-78.332,169.417,35.848,156.753
C08576=1042.213,-27.897,-78.345,169.419,35.848,156.753
C08577=1042.220,-27.647,-78.359,169.421,35.849,156.753
C08578=1042.226,-27.398,-78.372,169.423,35.850,156.753
C08579=1042.233,-27.148,-78.386,169.425,35.851,156.753
C08580=1042.239,-26.899,-78.399,169.427,35.852,156.753
C08581=1042.244,-26.649,-78.413,169.429,35.852,156.753
C08582=1042.251,-26.399,-78.426,169.431,35.853,156.753
C08583=1042.257,-26.150,-78.440,169.433,35.854,156.754
C08584=1042.263,-25.901,-78.454,169.436,35.855,156.754
C08585=1042.270,-25.651,-78.468,169.438,35.856,156.754
C08586=1042.276,-25.402,-78.481,169.440,35.856,156.754
C08587=1042.282,-25.151,-78.495,169.442,35.858,156.754
C08588=1042.288,-24.902,-78.509,169.445,35.858,156.754
C08589=1042.294,-24.653,-78.523,169.447,35.859,156.754
C08590=1042.301,-24.403,-78.537,169.449,35.860,156.754
C08591=1042.307,-24.154,-78.550,169.451,35.861,156.755
C08592=1042.313,-23.904,-78.564,169.453,35.862,156.755
C08593=1042.320,-23.654,-78.578,169.455,35.862,156.755
C08594=1042.326,-23.404,-78.591,169.457,35.864,156.755
C08595=1042.332,-23.156,-78.606,169.459,35.864,156.755
C08596=1042.338,-22.906,-78.619,169.461,35.865,156.755
C08597=1042.345,-22.656,-78.633,169.463,35.866,156.755
C08598=1042.351,-22.407,-78.647,169.465,35.867,156.756
C08599=1042.358,-22.157,-78.661,169.467,35.868,156.756
C08600=1042.363,-21.908,-78.675,169.469,35.868,156.756
C08601=1042.370,-21.658,-78.689,169.471,35.869,156.756
C08602=1042.376,-21.409,-78.702,169.473,35.870,156.756
C08603=1042.383,-21.159,-78.717,169.476,35.871,156.756
C08604=1042.389,-20.910,-78.730,169.478,35.872,156.756
C08605=1042.395,-20.659,-78.744,169.480,35.873,156.757
C08606=1042.401,-20.411,-78.758,169.482,35.874,156.757
C08607=1042.408,-20.161,-78.772,169.484,35.874,156.757
C08608=1042.414,-19.911,-78.786,169.486,35.875,156.757
C08609=1042.421,-19.629,-78.802,169.489,35.876,156.757
C08610=1042.428,-19.348,-78.818,169.491,35.877,156.757
C08611=1042.435,-19.066,-78.833,169.493,35.878,156.757
C08612=1042.443,-18.784,-78.849,169.496,35.879,156.758
C08613=1042.449,-18.535,-78.862,169.498,35.880,156.758
C08614=1042.456,-18.285,-78.877,169.500,35.881,156.758
C08615=1042.462,-18.036,-78.891,169.502,35.882,156.758
C08616=1042.468,-17.786,-78.905,169.504,35.882,156.758
C08617=1042.474,-17.537,-78.919,169.507,35.884,156.758
C08618=1042.480,-17.287,-78.933,169.509,35.884,156.758
C08619=1042.487,-17.038,-78.947,169.511,35.885,156.759
C08620=1042.494,-16.788,-78.961,169.513,35.886,156.759
C08621=1042.500,-16.538,-78.976,169.515,35.887,156.759
C08622=1042.506,-16.289,-78.989,169.517,35.888,156.759
C08623=1042.512,-16.039,-79.003,169.519,35.888,156.759
C08624=1042.519,-15.790,-79.017,169.521,35.890,156.759
C08625=1042.525,-15.540,-79.031,169.523,35.890,156.759
C08626=1042.532,-15.291,-79.045,169.525,35.891,156.760
C08627=1042.538,-15.041,-79.059,169.527,35.892,156.760
C08628=1042.545,-14.792,-79.074,169.529,35.893,156.760
C08629=1042.550,-14.542,-79.088,169.531,35.894,156.760
C08630=1042.557,-14.292,-79.103,169.533,35.895,156.760
C08631=1042.563,-14.043,-79.116,169.535,35.896,156.760
C08632=1042.569,-13.793,-79.131,169.538,35.897,156.761
C08633=1042.575,-13.545,-79.145,169.540,35.898,156.761
C08634=1042.582,-13.295,-79.159,169.542,35.899,156.761
C08635=1042.588,-13.045,-79.174,169.544,35.900,156.761
C08636=1042.594,-12.795,-79.188,169.546,35.900,156.761
C08637=1042.601,-12.546,-79.202,169.548,35.902,156.761
C08638=1042.607,-12.297,-79.217,169.549,35.902,156.761
C08639=1042.613,-12.047,-79.231,169.551,35.903,156.762
C08640=1042.620,-11.797,-79.245,169.553,35.904,156.762
C08641=1042.626,-11.548,-79.260,169.555,35.905,156.762
C08642=1042.632,-11.298,-79.274,169.557,35.906,156.762
C08643=1042.638,-11.050,-79.288,169.559,35.907,156.762
C08644=1042.644,-10.799,-79.302,169.562,35.908,156.762
C08645=1042.651,-10.550,-79.317,169.564,35.909,156.763
C08646=1042.657,-10.301,-79.331,169.566,35.910,156.763
C08647=1042.663,-10.051,-79.346,169.568,35.911,156.763
C08648=1042.670,-9.801,-79.361,169.570,35.912,156.763
C08649=1042.676,-9.552,-79.375,169.572,35.913,156.763
C08650=1042.683,-9.303,-79.389,169.574,35.914,156.763
C08651=1042.689,-9.052,-79.404,169.576,35.915,156.763
C08652=1042.695,-8.804,-79.418,169.578,35.915,156.764
C08653=1042.701,-8.554,-79.433,169.580,35.917,156.764
C08654=1042.708,-8.304,-79.447,169.582,35.917,156.764
C08655=1042.713,-8.055,-79.461,169.584,35.919,156.764
C08656=1042.720,-7.806,-79.476,169.586,35.919,156.764
C08657=1042.727,-7.556,-79.491,169.589,35.921,156.764
C08658=1042.733,-7.307,-79.505,169.591,35.921,156.765
C08659=1042.739,-7.057,-79.519,169.593,35.923,156.765
C08660=1042.746,-6.807,-79.534,169.595,35.923,156.765
C08661=1042.752,-6.558,-79.549,169.597,35.924,156.765
C08662=1042.758,-6.309,-79.563,169.599,35.925,156.765
C08663=1042.765,-6.059,-79.577,169.600,35.926,156.765
C08664=1042.771,-5.809,-79.592,169.602,35.927,156.766
C08665=1042.777,-5.560,-79.607,169.604,35.928,156.766
C08666=1042.784,-5.311,-79.621,169.606,35.929,156.766
C08667=1042.790,-5.061,-79.636,169.608,35.930,156.766
C08668=1042.797,-4.811,-79.651,169.610,35.930,156.766
C08669=1042.802,-4.562,-79.665,169.612,35.932,156.766
C08670=1042.809,-4.313,-79.679,169.615,35.932,156.766
C08671=1042.816,-4.063,-79.694,169.617,35.934,156.767
C08672=1042.822,-3.813,-79.709,169.619,35.934,156.767
C08673=1042.829,-3.530,-79.725,169.621,35.936,156.767
C08674=1042.837,-3.247,-79.742,169.623,35.937,156.767
C08675=1042.844,-2.963,-79.759,169.625,35.938,156.767
C08676=1042.850,-2.680,-79.776,169.628,35.939,156.768
C08677=1042.857,-2.431,-79.791,169.630,35.940,156.768
C08678=1042.863,-2.181,-79.806,169.631,35.942,156.768
C08679=1042.869,-1.932,-79.821,169.633,35.942,156.768
C08680=1042.875,-1.682,-79.836,169.635,35.944,156.768
C08681=1042.882,-1.433,-79.851,169.638,35.945,156.769
C08682=1042.888,-1.183,-79.866,169.640,35.945,156.769
C08683=1042.894,-0.934,-79.880,169.642,35.947,156.769
C08684=1042.900,-0.684,-79.895,169.644,35.947,156.769
C08685=1042.907,-0.435,-79.910,169.646,35.949,156.769
C08686=1042.913,-0.185,-79.925,169.648,35.950,156.769
C08687=1042.919,0.064,-79.940,169.649,35.951,156.770
C08688=1042.925,0.314,-79.955,169.651,35.952,156.770
C08689=1042.932,0.563,-79.970,169.653,35.953,156.770
C08690=1042.938,0.813,-79.985,169.655,35.954,156.770
C08691=1042.944,1.063,-79.999,169.658,35.955,156.770
C08692=1042.950,1.311,-80.014,169.660,35.957,156.771
C08693=1042.957,1.561,-80.029,169.662,35.957,156.771
C08694=1042.962,1.811,-80.045,169.664,35.959,156.771
C08695=1042.969,2.061,-80.059,169.666,35.959,156.771
C08696=1042.975,2.310,-80.075,169.667,35.960,156.771
C08697=1042.981,2.559,-80.090,169.669,35.962,156.771
C08698=1042.987,2.808,-80.105,169.671,35.962,156.772
C08699=1042.994,3.058,-80.120,169.673,35.964,156.772
C08700=1043.000,3.308,-80.135,169.675,35.965,156.772
C08701=1043.007,3.557,-80.150,169.677,35.966,156.772
C08702=1043.013,3.806,-80.165,169.680,35.967,156.772
C08703=1043.019,4.055,-80.180,169.682,35.968,156.772
C08704=1043.025,4.305,-80.195,169.683,35.969,156.773
C08705=1043.032,4.555,-80.210,169.685,35.970,156.773
C08706=1043.038,4.804,-80.225,169.687,35.971,156.773
C08707=1043.045,5.054,-80.240,169.689,35.972,156.773
C08708=1043.051,5.303,-80.256,169.691,35.973,156.773
C08709=1043.057,5.553,-80.271,169.693,35.974,156.774
C08710=1043.063,5.803,-80.286,169.695,35.975,156.774
C08711=1043.069,6.052,-80.300,169.697,35.976,156.774
C08712=1043.076,6.301,-80.316,169.698,35.977,156.774
C08713=1043.082,6.550,-80.331,169.701,35.979,156.774
C08714=1043.089,6.800,-80.346,169.703,35.979,156.775
C08715=1043.095,7.050,-80.361,169.705,35.981,156.775
C08716=1043.102,7.299,-80.376,169.707,35.982,156.775
C08717=1043.108,7.548,-80.391,169.709,35.983,156.775
C08718=1043.114,7.798,-80.407,169.711,35.984,156.775
C08719=1043.120,8.047,-80.423,169.713,35.985,156.775
C08720=1043.127,8.297,-80.438,169.714,35.986,156.776
C08721=1043.133,8.547,-80.452,169.716,35.987,156.776
C08722=1043.140,8.796,-80.468,169.718,35.988,156.776
C08723=1043.146,9.045,-80.483,169.720,35.989,156.776
C08724=1043.153,9.295,-80.498,169.723,35.990,156.776
C08725=1043.159,9.544,-80.514,169.725,35.991,156.777
C08726=1043.165,9.793,-80.528,169.727,35.992,156.777
C08727=1043.171,10.043,-80.544,169.728,35.993,156.777
C08728=1043.177,10.292,-80.559,169.730,35.994,156.777
C08729=1043.184,10.542,-80.574,169.732,35.996,156.777
C08730=1043.190,10.791,-80.589,169.734,35.996,156.777
C08731=1043.197,11.040,-80.605,169.736,35.998,156.778
C08732=1043.203,11.290,-80.620,169.738,35.998,156.778
C08733=1043.210,11.539,-80.636,169.740,36.000,156.778
C08734=1043.216,11.789,-80.651,169.741,36.001,156.778
C08735=1043.222,12.039,-80.666,169.744,36.001,156.778
C08736=1043.229,12.288,-80.682,169.746,36.003,156.779
C08737=1043.236,12.573,-80.699,169.748,36.004,156.779
C08738=1043.243,12.859,-80.716,169.750,36.005,156.779
C08739=1043.251,13.144,-80.734,169.753,36.006,156.779
C08740=1043.258,13.429,-80.752,169.755,36.007,156.779
C08741=1043.265,13.678,-80.767,169.757,36.009,156.780
C08742=1043.271,13.928,-80.782,169.758,36.009,156.780
C08743=1043.277,14.177,-80.799,169.760,36.011,156.780
C08744=1043.284,14.427,-80.814,169.762,36.012,156.780
C08745=1043.291,14.676,-80.829,169.765,36.013,156.780
C08746=1043.296,14.926,-80.845,169.767,36.014,156.780
C08747=1043.303,15.175,-80.860,169.769,36.015,156.781
C08748=1043.308,15.425,-80.876,169.770,36.016,156.781
C08749=1043.315,15.674,-80.892,169.772,36.018,156.781
C08750=1043.322,15.924,-80.907,169.774,36.018,156.781
C08751=1043.328,16.173,-80.923,169.776,36.020,156.781
C08752=1043.334,16.422,-80.939,169.778,36.021,156.782
C08753=1043.340,16.672,-80.954,169.779,36.022,156.782
C08754=1043.347,16.921,-80.970,169.781,36.023,156.782
C08755=1043.354,17.171,-80.986,169.784,36.024,156.782
C08756=1043.359,17.421,-81.001,169.786,36.025,156.782
C08757=1043.366,17.670,-81.017,169.788,36.027,156.783
C08758=1043.372,17.920,-81.032,169.790,36.027,156.783
C08759=1043.378,18.169,-81.048,169.791,36.029,156.783
C08760=1043.385,18.418,-81.064,169.793,36.030,156.783
C08761=1043.391,18.668,-81.079,169.795,36.031,156.784
C08762=1043.398,18.917,-81.095,169.797,36.032,156.784
C08763=1043.403,19.166,-81.111,169.799,36.033,156.784
C08764=1043.410,19.416,-81.126,169.801,36.034,156.784
C08765=1043.417,19.665,-81.142,169.803,36.035,156.784
C08766=1043.422,19.914,-81.158,169.805,36.036,156.784
C08767=1043.430,20.164,-81.174,169.807,36.038,156.785
C08768=1043.435,20.414,-81.190,169.809,36.039,156.785
C08769=1043.442,20.663,-81.205,169.810,36.040,156.785
C08770=1043.448,20.912,-81.222,169.812,36.041,156.785
C08771=1043.454,21.162,-81.238,169.814,36.042,156.785
C08772=1043.460,21.411,-81.253,169.816,36.043,156.786
C08773=1043.466,21.661,-81.269,169.818,36.045,156.786
C08774=1043.473,21.910,-81.285,169.820,36.046,156.786
C08775=1043.479,22.159,-81.301,169.822,36.047,156.786
C08776=1043.486,22.408,-81.317,169.824,36.048,156.786
C08777=1043.492,22.659,-81.333,169.826,36.049,156.787
C08778=1043.499,22.908,-81.348,169.828,36.051,156.787
C08779=1043.505,23.157,-81.364,169.829,36.052,156.787
C08780=1043.511,23.406,-81.380,169.831,36.053,156.787
C08781=1043.517,23.655,-81.396,169.833,36.054,156.787
C08782=1043.523,23.905,-81.413,169.835,36.055,156.788
C08783=1043.530,24.154,-81.428,169.837,36.056,156.788
C08784=1043.536,24.405,-81.444,169.839,36.058,156.788
C08785=1043.543,24.654,-81.460,169.841,36.059,156.788
C08786=1043.549,24.903,-81.476,169.843,36.060,156.788
C08787=1043.555,25.152,-81.492,169.845,36.061,156.789
C08788=1043.561,25.401,-81.508,169.846,36.062,156.789
C08789=1043.567,25.651,-81.524,169.848,36.063,156.789
C08790=1043.575,25.900,-81.540,169.850,36.064,156.789
C08791=1043.581,26.150,-81.557,169.852,36.065,156.790
C08792=1043.587,26.399,-81.572,169.854,36.067,156.790
C08793=1043.593,26.649,-81.588,169.856,36.068,156.790
C08794=1043.599,26.898,-81.604,169.858,36.069,156.790
C08795=1043.606,27.148,-81.620,169.860,36.071,156.790
C08796=1043.612,27.397,-81.636,169.862,36.071,156.791
C08797=1043.619,27.646,-81.652,169.863,36.072,156.791
C08798=1043.625,27.896,-81.668,169.865,36.074,156.791
C08799=1043.631,28.145,-81.685,169.867,36.075,156.791
C08800=1043.638,28.395,-81.701,169.869,36.076,156.791
C08801=1043.645,28.681,-81.720,169.871,36.078,156.792
C08802=1043.652,28.967,-81.738,169.874,36.079,156.792
C08803=1043.659,29.254,-81.756,169.876,36.080,156.792
C08804=1043.667,29.541,-81.775,169.878,36.081,156.792
C08805=1043.672,29.790,-81.791,169.880,36.083,156.793
C08806=1043.679,30.040,-81.808,169.881,36.084,156.793
C08807=1043.685,30.289,-81.824,169.883,36.085,156.793
C08808=1043.691,30.539,-81.840,169.885,36.087,156.793
C08809=1043.698,30.788,-81.856,169.887,36.088,156.794
C08810=1043.704,31.037,-81.873,169.889,36.089,156.794
C08811=1043.710,31.286,-81.890,169.891,36.090,156.794
C08812=1043.716,31.536,-81.906,169.893,36.092,156.794
C08813=1043.722,31.785,-81.922,169.895,36.092,156.794
C08814=1043.730,32.035,-81.938,169.896,36.094,156.795
C08815=1043.736,32.284,-81.954,169.898,36.095,156.795
C08816=1043.742,32.534,-81.971,169.900,36.096,156.795
C08817=1043.747,32.783,-81.987,169.902,36.097,156.795
C08818=1043.754,33.032,-82.004,169.903,36.099,156.795
C08819=1043.761,33.281,-82.020,169.906,36.100,156.796
C08820=1043.767,33.531,-82.036,169.908,36.101,156.796
C08821=1043.773,33.780,-82.052,169.910,36.103,156.796
C08822=1043.779,34.030,-82.069,169.911,36.103,156.796
C08823=1043.786,34.279,-82.086,169.913,36.105,156.796
C08824=1043.792,34.528,-82.102,169.915,36.106,156.797
C08825=1043.799,34.778,-82.118,169.917,36.107,156.797
C08826=1043.805,35.027,-82.135,169.918,36.108,156.797
C08827=1043.811,35.277,-82.151,169.920,36.110,156.797
C08828=1043.818,35.526,-82.168,169.923,36.111,156.798
C08829=1043.824,35.775,-82.184,169.925,36.112,156.798
C08830=1043.830,36.025,-82.201,169.926,36.113,156.798
C08831=1043.837,36.275,-82.217,169.928,36.114,156.798
C08832=1043.843,36.523,-82.234,169.930,36.115,156.798
C08833=1043.849,36.773,-82.250,169.932,36.117,156.799
C08834=1043.856,37.023,-82.267,169.933,36.118,156.799
C08835=1043.862,37.271,-82.284,169.935,36.119,156.799
C08836=1043.868,37.521,-82.300,169.938,36.121,156.799
C08837=1043.874,37.771,-82.316,169.940,36.122,156.800
C08838=1043.880,38.020,-82.333,169.941,36.123,156.800
C08839=1043.887,38.269,-82.350,169.943,36.124,156.800
C08840=1043.893,38.519,-82.366,169.945,36.126,156.800
C08841=1043.899,38.768,-82.383,169.946,36.127,156.801
C08842=1043.905,39.017,-82.400,169.948,36.128,156.801
C08843=1043.912,39.267,-82.416,169.950,36.129,156.801
C08844=1043.918,39.516,-82.433,169.953,36.131,156.801
C08845=1043.924,39.765,-82.449,169.954,36.132,156.801
C08846=1043.931,40.015,-82.467,169.956,36.133,156.802
C08847=1043.937,40.264,-82.483,169.958,36.134,156.802
C08848=1043.944,40.514,-82.500,169.959,36.135,156.802
C08849=1043.950,40.763,-82.517,169.961,36.137,156.802
C08850=1043.956,41.012,-82.533,169.963,36.138,156.802
C08851=1043.963,41.261,-82.550,169.965,36.139,156.803
C08852=1043.969,41.511,-82.566,169.966,36.140,156.803
C08853=1043.974,41.760,-82.584,169.969,36.142,156.803
C08854=1043.981,42.010,-82.601,169.971,36.143,156.803
C08855=1043.987,42.259,-82.618,169.973,36.144,156.804
C08856=1043.993,42.509,-82.634,169.974,36.145,156.804
C08857=1043.999,42.758,-82.650,169.976,36.147,156.804
C08858=1044.006,43.007,-82.667,169.978,36.148,156.804
C08859=1044.012,43.256,-82.685,169.979,36.149,156.805
C08860=1044.018,43.506,-82.701,169.981,36.151,156.805
C08861=1044.025,43.755,-82.718,169.984,36.152,156.805
C08862=1044.031,44.005,-82.735,169.986,36.153,156.805
C08863=1044.037,44.253,-82.752,169.987,36.154,156.805
C08864=1044.043,44.503,-82.769,169.989,36.156,156.806
C08865=1044.050,44.789,-82.789,169.991,36.158,156.806
C08866=1044.057,45.076,-82.808,169.993,36.159,156.806
C08867=1044.064,45.363,-82.828,169.995,36.161,156.807
C08868=1044.071,45.649,-82.848,169.998,36.162,156.807
C08869=1044.077,45.898,-82.865,169.999,36.163,156.807
C08870=1044.084,46.148,-82.881,170.001,36.165,156.807
C08871=1044.089,46.397,-82.899,170.003,36.166,156.808
C08872=1044.096,46.647,-82.915,170.004,36.167,156.808
C08873=1044.102,46.896,-82.932,170.006,36.169,156.808
C08874=1044.108,47.145,-82.950,170.008,36.170,156.808
C08875=1044.114,47.395,-82.967,170.010,36.172,156.809
C08876=1044.121,47.644,-82.983,170.012,36.173,156.809
C08877=1044.127,47.893,-83.001,170.014,36.174,156.809
C08878=1044.133,48.142,-83.018,170.016,36.175,156.809
C08879=1044.140,48.392,-83.035,170.017,36.177,156.810
C08880=1044.145,48.641,-83.053,170.019,36.178,156.810
C08881=1044.152,48.891,-83.070,170.021,36.179,156.810
C08882=1044.158,49.140,-83.086,170.022,36.180,156.810
C08883=1044.164,49.390,-83.104,170.024,36.182,156.810
C08884=1044.170,49.638,-83.121,170.027,36.183,156.811
C08885=1044.177,49.888,-83.138,170.028,36.184,156.811
C08886=1044.182,50.137,-83.155,170.030,36.186,156.811
C08887=1044.189,50.387,-83.173,170.032,36.187,156.811
C08888=1044.195,50.636,-83.190,170.033,36.189,156.812
C08889=1044.202,50.885,-83.208,170.035,36.190,156.812
C08890=1044.208,51.135,-83.224,170.037,36.191,156.812
C08891=1044.214,51.384,-83.242,170.040,36.193,156.812
C08892=1044.220,51.633,-83.259,170.041,36.194,156.813
C08893=1044.227,51.883,-83.276,170.043,36.195,156.813
C08894=1044.232,52.132,-83.294,170.045,36.196,156.813
C08895=1044.239,52.382,-83.310,170.046,36.198,156.813
C08896=1044.245,52.630,-83.327,170.048,36.199,156.814
C08897=1044.251,52.880,-83.345,170.050,36.200,156.814
C08898=1044.257,53.129,-83.362,170.051,36.201,156.814
C08899=1044.264,53.378,-83.379,170.054,36.203,156.814
C08900=1044.270,53.627,-83.397,170.056,36.204,156.814
C08901=1044.277,53.877,-83.414,170.058,36.205,156.815
C08902=1044.282,54.126,-83.431,170.059,36.207,156.815
C08903=1044.289,54.376,-83.449,170.061,36.208,156.815
C08904=1044.296,54.625,-83.466,170.063,36.209,156.815
C08905=1044.301,54.874,-83.483,170.064,36.210,156.816
C08906=1044.308,55.124,-83.501,170.066,36.212,156.816
C08907=1044.314,55.373,-83.518,170.069,36.213,156.816
C08908=1044.320,55.622,-83.536,170.070,36.215,156.816
C08909=1044.327,55.872,-83.553,170.072,36.216,156.817
C08910=1044.333,56.121,-83.571,170.074,36.217,156.817
C08911=1044.340,56.370,-83.588,170.075,36.219,156.817
C08912=1044.346,56.619,-83.605,170.077,36.220,156.817
C08913=1044.352,56.869,-83.622,170.079,36.221,156.818
C08914=1044.359,57.119,-83.639,170.082,36.222,156.818
C08915=1044.364,57.368,-83.657,170.083,36.224,156.818
C08916=1044.371,57.617,-83.674,170.085,36.225,156.818
C08917=1044.377,57.866,-83.691,170.087,36.226,156.819
C08918=1044.383,58.116,-83.709,170.088,36.227,156.819
C08919=1044.390,58.365,-83.727,170.090,36.229,156.819
C08920=1044.396,58.614,-83.744,170.092,36.230,156.819
C08921=1044.403,58.863,-83.761,170.093,36.231,156.819
C08922=1044.409,59.113,-83.779,170.096,36.233,156.820
C08923=1044.415,59.362,-83.796,170.098,36.234,156.820
C08924=1044.422,59.611,-83.814,170.100,36.235,156.820
C08925=1044.428,59.861,-83.832,170.101,36.236,156.820
C08926=1044.434,60.109,-83.849,170.103,36.238,156.821
C08927=1044.441,60.359,-83.867,170.105,36.239,156.821
C08928=1044.447,60.608,-83.885,170.106,36.240,156.821
C08929=1044.454,60.894,-83.905,170.108,36.241,156.821
C08930=1044.462,61.181,-83.925,170.111,36.243,156.822
C08931=1044.469,61.467,-83.945,170.113,36.245,156.822
C08932=1044.476,61.754,-83.965,170.115,36.246,156.822
C08933=1044.483,62.002,-83.982,170.117,36.247,156.822
C08934=1044.489,62.252,-84.000,170.119,36.248,156.823
C08935=1044.496,62.501,-84.017,170.120,36.250,156.823
C08936=1044.503,62.751,-84.035,170.122,36.251,156.823
C08937=1044.508,62.999,-84.053,170.125,36.252,156.823
C08938=1044.515,63.249,-84.070,170.126,36.253,156.824
C08939=1044.521,63.498,-84.088,170.128,36.255,156.824
C08940=1044.528,63.748,-84.106,170.130,36.256,156.824
C08941=1044.534,63.997,-84.123,170.131,36.257,156.824
C08942=1044.541,64.246,-84.141,170.133,36.259,156.824
C08943=1044.547,64.495,-84.159,170.135,36.260,156.825
C08944=1044.553,64.745,-84.177,170.136,36.261,156.825
C08945=1044.559,64.994,-84.194,170.139,36.262,156.825
C08946=1044.566,65.244,-84.212,170.141,36.264,156.825
C08947=1044.572,65.493,-84.231,170.143,36.266,156.826
C08948=1044.578,65.742,-84.248,170.144,36.267,156.826
C08949=1044.584,65.991,-84.266,170.146,36.268,156.826
C08950=1044.590,66.241,-84.284,170.148,36.269,156.826
C08951=1044.596,66.489,-84.302,170.149,36.271,156.827
C08952=1044.603,66.739,-84.319,170.152,36.272,156.827
C08953=1044.609,66.989,-84.337,170.154,36.273,156.827
C08954=1044.616,67.238,-84.356,170.155,36.274,156.827
C08955=1044.622,67.486,-84.373,170.157,36.276,156.828
C08956=1044.628,67.736,-84.391,170.159,36.278,156.828
C08957=1044.634,67.985,-84.409,170.160,36.279,156.828
C08958=1044.641,68.235,-84.427,170.162,36.280,156.828
C08959=1044.646,68.484,-84.445,170.165,36.281,156.829
C08960=1044.653,68.733,-84.463,170.166,36.283,156.829
C08961=1044.659,68.983,-84.481,170.168,36.284,156.829
C08962=1044.666,69.232,-84.499,170.170,36.285,156.829
C08963=1044.672,69.482,-84.517,170.171,36.286,156.830
C08964=1044.678,69.730,-84.534,170.173,36.288,156.830
C08965=1044.685,69.979,-84.553,170.175,36.290,156.830
C08966=1044.691,70.229,-84.571,170.177,36.291,156.830
C08967=1044.697,70.479,-84.589,170.179,36.292,156.831
C08968=1044.703,70.727,-84.607,170.181,36.293,156.831
C08969=1044.709,70.977,-84.625,170.182,36.295,156.831
C08970=1044.715,71.226,-84.644,170.184,36.296,156.832
C08971=1044.721,71.476,-84.662,170.186,36.298,156.832
C08972=1044.728,71.724,-84.679,170.187,36.299,156.832
C08973=1044.734,71.974,-84.697,170.190,36.300,156.832
C08974=1044.740,72.223,-84.716,170.192,36.301,156.832
C08975=1044.747,72.473,-84.734,170.193,36.303,156.833
C08976=1044.753,72.722,-84.752,170.195,36.305,156.833
C08977=1044.759,72.971,-84.770,170.197,36.306,156.833
C08978=1044.765,73.220,-84.789,170.198,36.307,156.834
C08979=1044.771,73.470,-84.807,170.200,36.308,156.834
C08980=1044.778,73.719,-84.825,170.203,36.310,156.834
C08981=1044.784,73.969,-84.843,170.204,36.312,156.834
C08982=1044.790,74.218,-84.862,170.206,36.313,156.835
C08983=1044.796,74.467,-84.879,170.208,36.314,156.835
C08984=1044.802,74.716,-84.898,170.209,36.315,156.835
C08985=1044.809,74.965,-84.916,170.211,36.317,156.835
C08986=1044.815,75.214,-84.934,170.213,36.318,156.836
C08987=1044.822,75.463,-84.953,170.215,36.320,156.836
C08988=1044.828,75.713,-84.971,170.217,36.321,156.836
C08989=1044.834,75.962,-84.989,170.219,36.322,156.836
C08990=1044.840,76.211,-85.008,170.220,36.324,156.837
C08991=1044.846,76.460,-85.025,170.222,36.325,156.837
C08992=1044.853,76.710,-85.044,170.224,36.326,156.837
C08993=1044.860,76.996,-85.066,170.226,36.328,156.837
C08994=1044.867,77.282,-85.086,170.229,36.329,156.838
C08995=1044.874,77.568,-85.107,170.230,36.331,156.838
C08996=1044.881,77.853,-85.128,170.232,36.332,156.838
C08997=1044.888,78.103,-85.147,170.234,36.334,156.839
C08998=1044.894,78.352,-85.165,170.236,36.335,156.839
C08999=1044.900,78.601,-85.183,170.237,36.337,156.839
C09000=1044.906,78.851,-85.202,170.240,36.338,156.839
C09001=1044.912,79.100,-85.221,170.242,36.340,156.840
C09002=1044.918,79.350,-85.239,170.243,36.341,156.840
C09003=1044.924,79.598,-85.257,170.245,36.342,156.840
C09004=1044.931,79.847,-85.276,170.247,36.344,156.840
C09005=1044.936,80.097,-85.295,170.248,36.346,156.841
C09006=1044.943,80.346,-85.314,170.250,36.347,156.841
C09007=1044.949,80.596,-85.332,170.253,36.348,156.841
C09008=1044.955,80.845,-85.350,170.254,36.349,156.841
C09009=1044.962,81.094,-85.369,170.256,36.351,156.842
C09010=1044.967,81.343,-85.388,170.258,36.352,156.842
C09011=1044.974,81.592,-85.407,170.259,36.354,156.842
C09012=1044.979,81.841,-85.425,170.261,36.355,156.842
C09013=1044.986,82.091,-85.443,170.264,36.357,156.843
C09014=1044.992,82.340,-85.462,170.265,36.358,156.843
C09015=1044.998,82.589,-85.481,170.267,36.359,156.843
C09016=1045.004,82.838,-85.500,170.269,36.361,156.844
C09017=1045.011,83.087,-85.518,170.270,36.363,156.844
C09018=1045.017,83.337,-85.536,170.272,36.364,156.844
C09019=1045.023,83.586,-85.555,170.274,36.365,156.844
C09020=1045.029,83.836,-85.574,170.276,36.366,156.845
C09021=1045.035,84.085,-85.593,170.278,36.368,156.845
C09022=1045.042,84.334,-85.612,170.280,36.369,156.845
C09023=1045.048,84.583,-85.630,170.281,36.371,156.845
C09024=1045.054,84.832,-85.649,170.283,36.372,156.846
C09025=1045.060,85.082,-85.668,170.285,36.374,156.846
C09026=1045.067,85.331,-85.687,170.287,36.375,156.846
C09027=1045.073,85.580,-85.705,170.289,36.376,156.846
C09028=1045.080,85.829,-85.724,170.291,36.378,156.847
C09029=1045.085,86.078,-85.743,170.292,36.379,156.847
C09030=1045.092,86.328,-85.762,170.294,36.381,156.847
C09031=1045.098,86.577,-85.780,170.296,36.382,156.848
C09032=1045.104,86.826,-85.799,170.297,36.383,156.848
C09033=1045.110,87.076,-85.818,170.300,36.384,156.848
C09034=1045.116,87.325,-85.836,170.302,36.386,156.848
C09035=1045.123,87.574,-85.855,170.303,36.388,156.849
C09036=1045.129,87.823,-85.874,170.305,36.389,156.849
C09037=1045.135,88.073,-85.893,170.307,36.390,156.849
C09038=1045.141,88.322,-85.912,170.308,36.391,156.849
C09039=1045.148,88.571,-85.930,170.310,36.393,156.850
C09040=1045.155,88.819,-85.950,170.313,36.395,156.850
C09041=1045.160,89.069,-85.969,170.314,36.396,156.850
